// TwinCAT 3 PLC project ApplicationBase
// Title: ApplicationBase
// Company: Beckhoff Automation LLC
// Author: FS
// ProjectVersion: 2.3.0
// Description: All sample code provided by Beckhoff Automation LLC are for illustrative purposes only and are provided “as is” and without any warranties, express or implied. Actual implementations in applications will vary significantly. Beckhoff Automation LLC shall have no liability for, and does not waive any rights in relation to, any code samples that it provides or the use of such code samples for any purpose.
// ProgramVersion: 3.1.4026.27
// libraries:
//   Tc2_DataExchange, * (Beckhoff Automation GmbH)
//   Tc2_EtherCAT, * (Beckhoff Automation GmbH)
//   Tc2_IoFunctions, * (Beckhoff Automation GmbH)
//   Tc2_Math, * (Beckhoff Automation GmbH)
//   Tc2_MC2, * (Beckhoff Automation GmbH)
//   Tc2_MC2_Camming, * (Beckhoff Automation GmbH)
//   Tc2_MC2_Drive, * (Beckhoff Automation GmbH)
//   Tc2_NcKinematicTransformation, * (Beckhoff Automation GmbH)
//   Tc2_SerialCom, * (Beckhoff Automation GmbH)
//   Tc2_Standard, * (Beckhoff Automation GmbH)
//   Tc2_System, * (Beckhoff Automation GmbH)
//   Tc2_TcpIp, * (Beckhoff Automation GmbH)
//   Tc2_Utilities, * (Beckhoff Automation GmbH)
//   Tc3_DynamicMemory, * (Beckhoff Automation GmbH)
//   Tc3_EventLogger, * (Beckhoff Automation GmbH)
//   Tc3_JsonXml, * (Beckhoff Automation GmbH)
//   Tc3_MC2_AdvancedHoming, * (Beckhoff Automation GmbH)
//   Tc3_Mc3Ptp, * (Beckhoff Automation GmbH)
//   Tc3_Module, * (Beckhoff Automation GmbH)
//   Tc3_PackML_V3, * (Beckhoff Automation GmbH)
// project tree:
//   Components/ADS/ AdsReadWrite.TcPOU
//   Components/ADS/Interface/ I_AdsAccess.TcIO, I_AdsRW.TcIO
//   Components/Analog/ AnalogInput.TcPOU, AnalogInput_Generic.TcPOU, AnalogInput_Standard.TcPOU, AnalogOutput.TcPOU
//   Components/Analog/DUT/ ST_AnalogInputStatus_EL30xx.TcDUT, ST_AnalogInputStatus_Generic.TcDUT
//   Components/Analog/Interface/ I_AnalogChannel_Generic.TcIO, I_AnalogChannel_Standard.TcIO, I_AnalogInput.TcIO, I_AnalogOutput.TcIO
//   Components/CoE/ CoeDevice.TcPOU, NullCoeDevice.TcPOU
//   Components/CoE/DUT/ ST_TerminalProductInfo.TcDUT
//   Components/CoE/Interface/ I_CoeAccess.TcIO, I_CoeDevice.TcIO, I_CoeTransfer.TcIO, I_CoeTransferScheduler.TcIO
//   Components/Cylinder/ Cylinder.TcPOU, Cylinder_HMI.TcPOU, Cylinder_TcEvents.TcPOU
//   Components/Cylinder/DUT/ E_CylinderErrorId.TcDUT, E_CylinderState.TcDUT, ST_Cylinder_HMI.TcDUT
//   Components/Cylinder/Interface/ I_Cylinder.TcIO, I_CylinderCommand.TcIO, I_CylinderStatus.TcIO
//   Components/Digital/ DigitalInput_Combiner.TcPOU, DigitalInput_DebounceFallingEdge.TcPOU, DigitalInput_DebounceRisingEdge.TcPOU, DigitalInput_HMI.TcPOU, DigitalInput_NC.TcPOU, DigitalInput_NO.TcPOU, DigitalOutput.TcPOU, DigitalOutput_HMI.TcPOU
//   Components/Digital/DUT/ ST_DigitalInput_HMI.TcDUT, ST_DigitalOutput_HMI.TcDUT
//   Components/Digital/Interface/ I_DigitalInput.TcIO, I_DigitalOutput.TcIO
//   Components/Digital/Visitor/ ForceVisitor.TcPOU, ReleaseAllForceVisitor.TcPOU
//   Components/EtherCat/DUT/ E_EcErrorSource.TcDUT, EtherCatParameter.TcGVL, ST_EtherCatMasterInfo.TcDUT, ST_EtherCatSyncUnitTaskInfo.TcDUT
//   Components/EtherCat/ EtherCatIoDevice.TcPOU, EtherCatMaster.TcPOU, EtherCatMaster_TcEvents.TcPOU, SyncUnitTask.TcPOU
//   Components/EtherCat/Interface/ I_EcIoDevice.TcIO, I_EcSlaveRegistry.TcIO, I_EtherCatDiagnosticEventProvider.TcIO, I_EtherCatMasterDiagnostic.TcIO, I_IoDevice.TcIO, I_SyncUnitTask.TcIO
//   Components/Recipe/Interface/ I_RecipeManagment.TcIO
//   Components/Recipe/ RecipeManagment.TcPOU
//   Components/Safety/DUT/ E_SafetyConnection_State.TcDUT, E_SafetyEdm_State.TcDUT, E_SafetyEStop_State.TcDUT, E_SafetyGroup_Diag.TcDUT, E_SafetyGroup_State.TcDUT, E_SafetyMon_State.TcDUT, E_SafetyOrAnd_State.TcDUT, ST_SafetyAddressInfo.TcDUT, ST_SafetyDeviceInfo.TcDUT, ST_SafetyStateDiag.TcDUT
//   Components/Safety/Interface/ I_InSafetyGroup.TcIO, I_SafetyBase.TcIO, I_SafetyModule.TcIO, I_SafetyReset.TcIO, I_SafetySimulation.TcIO
//   Components/Safety/Reset Function/ SafetyResetPulse.TcPOU
//   Components/Safety/ SafetyAndOrFB.TcPOU, SafetyBase.TcPOU, SafetyConnectionFB_TcEvents.TcPOU, SafetyEdmFB_TcEvents.TcPOU, SafetyEstopFB_TcEvents.TcPOU, SafetyGroup_TcEvents.TcPOU, SafetyModule.TcPOU, SafetyMonFB_TcEvents.TcPOU
//   Components/Safety/Visitor/ SafetyOkVisitor.TcPOU, SetSafetySimulationVisitor.TcPOU
//   Components/Serial/Interface/ I_SerialByteConnection.TcIO, I_SerialLineControl.TcIO, I_SerialStringConnection.TcIO
//   Components/Serial/ SerialByteConnection.TcPOU, SerialLineControl_ADS.TcPOU, SerialLineControl_Terminal.TcPOU, SerialStringConnection.TcPOU
//   Components/Tcp Ip/DUT/ ST_TcpIpPayload.TcDUT
//   Components/Tcp Ip/Interface/ I_TcpIpConnection.TcIO, I_TcpIpSubscription.TcIO
//   Components/Tcp Ip/ TcpIpCommandResultFilter.TcPOU, TcpIpConnection.TcPOU, TcpIpConnectionParameter.TcGVL
//   Component/ Component.TcPOU, CyclicComponent.TcPOU
//   Component/Interface/ I_Component.TcIO, I_ComponentVisitor.TcIO
//   / ApplicationBaseParameter.TcGVL, ApplicationBaseMotionParameter.TcGVL
//   Events/Interface/ I_EventArguments.TcIO, I_EventClass.TcIO, I_EventClassTcEvents.TcIO, I_EventReaction.TcIO, I_EventReactionTcEvents.TcIO
//   Events/ TcEventClass.TcPOU
//   HMI/ Button.TcPOU, HmiFunction.TcPOU
//   HMI/DUT/ ST_HmiFunction.TcDUT
//   HMI/Interface/ I_Button.TcIO, I_HmiFunction.TcIO, I_Permissive.TcIO, I_StringCollection.TcIO
//   Kinematic Group/Interface/ I_KinematicGroup.TcIO
//   Kinematic Group/ KinematicGroup.TcPOU, KinematicGroup_TcEvents.TcPOU
//   Modes/Interface/ I_Mode.TcIO
//   Modes/ ModeControl.TcPOU, PackMLModeControl.TcPOU
//   Module PackML/ PackMLModule.TcPOU
//   Module/Interface/ I_Module.TcIO, I_ModuleVisitor.TcIO
//   Module/ Module.TcPOU
//   Motion/ AxisPTP_HMI.TcPOU, Axis_TcEvents.TcPOU
//   Motion/DUT/ E_AxisJogMode.TcDUT, ST_AxisPTP_HMI.TcDUT, ST_NcAxisStatus.TcDUT
//   Motion/Interface/ I_AxisDynamics.TcIO, I_AxisEnable.TcIO, I_AxisHome.TcIO, I_AxisJog.TcIO, I_AxisMoveAbsolute.TcIO, I_AxisMoveModulo.TcIO, I_AxisMoveRelative.TcIO, I_AxisMoveVelocity.TcIO, I_AxisStatus.TcIO, I_Axis.TcIO, I_AxisGear.TcIO, I_AxisSettings.TcIO, I_Axis_PTP.TcIO, I_MotionTaskCollection.TcIO
//   Motion/MC2/DUT/ ST_Mc2MotionDefaults.TcDUT
//   Motion/MC2/Interface/ I_Mc2Axis.TcIO, I_Mc2AxisGear.TcIO, I_Mc2Axis_PTP.TcIO, I_Mc2Settings.TcIO, I_Mc2SlaveAxis.TcIO
//   Motion/MC2/ Mc2Axis.TcPOU, Mc2AxisPTP.TcPOU, Mc2AxisParameterLoader.TcPOU, Mc2SlaveAxisPTP.TcPOU
//   Motion/MC3/DUT/ ST_Mc3MotionDefaults.TcDUT, ST_Mc3ParameterBinding.TcDUT
//   Motion/MC3/Interface/ I_Mc3SlaveAxis.TcIO, I_Mc3AxisGear.TcIO, I_Mc3Axis_PTP.TcIO, I_Mc3Settings.TcIO, I_Mc3Axis.TcIO
//   Motion/MC3/ Mc3SlaveAxisPTP.TcPOU, Mc3AxisPTP.TcPOU, Mc3AxisParameterLoader.TcPOU, Mc3Axis.TcPOU
//   Permissive Interlock/ PermissiveInterlock.TcPOU
//   Project Information/ F_GetCompany.TcPOU, F_GetTitle.TcPOU, F_GetVersion.TcPOU
//   Statemachine/DUT/ ST_PackMLStatemachine_HMI.TcDUT, ST_Statemachine_HMI.TcDUT
//   Statemachine/Generic/ NextMinorStep.TcPOU (not stored), NextStep.TcPOU (not stored), SetStep.TcPOU (not stored), State.TcPOU, Statemachine.TcPOU, Statemachine_HMI.TcPOU
//   Statemachine/Interface/ I_ContainStatemachine.TcIO, I_State.TcIO, I_Statemachine.TcIO
//   Statemachine/PackML/ NextAvailablePackMLCommands.TcPOU (not stored), PackMLStatemachine.TcPOU, PackMLStatemachine_HMI.TcPOU, PackMLStatemachine_ModuleIntegrated.TcPOU
//   Tracing/ CoreTrace.TcGVL, Trace.TcPOU
//   Tracing/DUT/ TcEventSeverityExt.TcDUT (not stored)
//   Tracing/Interface/ I_Trace.TcIO (not stored)
//   Utilities/AnyBuffer/ AnyBuffer.TcPOU
//   Utilities/AnyBuffer/DUT/ ST_BufferConfiguration.TcDUT, ST_BufferMetadata.TcDUT
//   Utilities/AnyBuffer/Interface/ I_AnyBuffer.TcIO, I_AnyBufferStrategy.TcIO
//   Utilities/AnyBuffer/TypedBuffers/ FifoBuffer.TcPOU, LifoBuffer.TcPOU, ListBuffer.TcPOU, RingBuffer.TcPOU
//   Utilities/File/DUT/ ST_File_HMI.TcDUT
//   Utilities/File/ File_HMI.TcPOU, JsonFile.TcPOU, StringHelper.TcPOU
//   Utilities/File/Interface/ I_FileHandler.TcIO
//   Utilities/Flash/ SyncedSquareWaves.TcPOU
//   Utilities/Force/DUT/ E_ForceState.TcDUT
//   Utilities/Force/ ForcibleBool.TcPOU, ForcibleInt.TcPOU
//   Utilities/Force/Interface/ I_ForcibleBool.TcIO, I_ForcibleInt.TcIO
//   Utilities/Functions/ CompareLREAL.TcPOU, CompareModulo.TcPOU, PercentToAnalog.TcPOU
//   Utilities/Motion/ ATAN2.TcPOU, CalculateHypotenuseAngle.TcPOU, CalculateMotionDynamics.TcPOU, CamSmoothError.TcDUT, CamSplineBoundary.TcDUT, CamSmoothDerivatives.TcPOU, MotionDynamicsError.TcDUT, XPlanar6DMoverToWorldTransform.TcPOU
//   Utilities/Scaling/ AnalogScale.TcPOU, Calibrate.TcPOU
//   Utilities/Scaling/Interface/ I_AnalogScalable.TcIO, I_AnalogScale.TcIO, I_CalibratableLinear.TcIO, I_CalibrateLinear.TcIO, I_TransformLRealValue.TcIO
//   Utilities/Timing/ Stopwatch.TcPOU
//   Version/ Global_Version.TcGVL
//   Visitors/Enable/ CheckComponentsEnabledVisitor.TcPOU, DisableAllComponentsVisitor.TcPOU, EnableAllComponentsVisitor.TcPOU
//   Visitors/Events/ GetActiveEventSeverityVisitor.TcPOU
//   Visitors/HMI/ GetSystemTreeJsonHmiVisitor.TcPOU, HmiEnableDisableAllVisitor.TcPOU
//   Visitors/Override/ SetAllOverrideVisitor.TcPOU
//   Visitors/PackML Statemachine/ ChangePackMLStateOnAllSubModulesVisitor.TcPOU, EventReactorPackMLVisitor.TcPOU
//   Visitors/Reset/ GetComponentsTaskResultVisitor.TcPOU, ResetAllVisitor.TcPOU, ResetComponentsVisitor.TcPOU, ResetModulesVisitor.TcPOU
//   Visitors/Statemachine/ ChangeModeOnAllSubModulesVisitor.TcPOU, ChangeStateOnAllSubModulesVisitor.TcPOU, EventReactorVisitor.TcPOU
//   Visitors/Stop/ StopAllComponentsVisitor.TcPOU
//   _Interface/ I_Base.TcIO (not stored), I_Command.TcIO, I_Disposable.TcIO, I_Enablable.TcIO, I_Initializable.TcIO, I_Override.TcIO, I_Resettable.TcIO, I_Simulatable.TcIO, I_Stoppable.TcIO, I_TaskResult.TcIO, I_ToString.TcIO (not stored)
//   _Internal/CollectionPeeker/ CollectionPeeker.TcPOU
//   _Internal/CollectionPeeker/Interface/ I_CollectionPeeker.TcIO, I_Peekable.TcIO, I_Peeker.TcIO
//   _Internal/Collection/ Collection.TcPOU
//   _Internal/Collection/Interface/ I_Collection.TcIO, I_Enumerator.TcIO
//   _Internal/Component/ ComponentCollection.TcPOU
//   _Internal/Component/Interface/ I_ComponentCollection.TcIO, I_ContainComponents.TcIO
//   _Internal/Cyclic/ CyclicRunner.TcPOU
//   _Internal/Cyclic/Interface/ I_Cyclic.TcIO
//   _Internal/Events/ TcEventClassArguments.TcPOU
//   _Internal/Initialize/ Initializer.TcPOU
//   _Internal/List/Interface/ I_List.TcIO
//   _Internal/List/ List.TcPOU
//   _Internal/Module/Interface/ I_ContainModules.TcIO, I_ModuleCollection.TcIO
//   _Internal/Module/ ModuleCollection.TcPOU
//   _Internal/MotionTasks/DUT/ ST_TaskState.TcDUT
//   _Internal/MotionTasks/MC2/AX5000/DUT/P_0_0074/ ST_IDN_P_0_0074.TcDUT (not stored), ST_IDN_P_0_0074_UDINT.TcDUT
//   _Internal/MotionTasks/MC2/AX5000/DUT/P_0_0074_LREAL/ ST_IDN_P_0_0074_LREAL.TcDUT
//   _Internal/MotionTasks/MC2/AX5000/DUT/ ST_AX5000AmpToNm.TcDUT
//   _Internal/MotionTasks/MC2/AX5000/ Mc2MotionTask_AX5000AmpToNm.TcPOU
//   _Internal/MotionTasks/MC2/Base/ Mc2MotionTask.TcPOU, Mc2MotionTaskCollection.TcPOU
//   _Internal/MotionTasks/MC2/Coupling/ Mc2MotionCoupleTask_Gearing.TcPOU
//   _Internal/MotionTasks/MC2/Home/ Mc2MotionHomeTask_CoESetEncoderOffset.TcPOU, Mc2MotionHomeTask_SetPosition.TcPOU, Mc2MotionHomeTask_SetPositionOffset.TcPOU, Mc2MotionHomeTask_SetZeroHere.TcPOU, Mc2MotionHomeTask_TouchProbe.TcPOU
//   _Internal/MotionTasks/MC2/Interface/ I_Mc2AxisRef.TcIO, I_Mc2MotionJogTask.TcIO, I_Mc2MotionPowerTask.TcIO, I_Mc2MotionTask.TcIO, I_Mc2MotionTaskCollection.TcIO
//   _Internal/MotionTasks/MC2/Move/ Mc2MoveAbsoluteTask.TcPOU, Mc2MoveJogTask.TcPOU, Mc2MoveModuloTask.TcPOU, Mc2MoveRelativeTask.TcPOU, Mc2MoveVelocityTask.TcPOU
//   _Internal/MotionTasks/MC2/Power/ Mc2PowerTask.TcPOU, Mc2StopTask.TcPOU
//   _Internal/MotionTasks/MC2/Reset/ Mc2CoEExtendedResetTask.TcPOU, Mc2CoEResetTask.TcPOU, Mc2SoEResetTask.TcPOU
//   _Internal/MotionTasks/MC3/Base/ Mc3MotionTaskCollection.TcPOU, Mc3MotionTask.TcPOU
//   _Internal/MotionTasks/MC3/Gearing/ Mc3MotionCoupleTask_Gearing.TcPOU
//   _Internal/MotionTasks/MC3/Home/ Mc3MotionHomeTask_SetPosition.TcPOU, Mc3MotionHomeTask_SetZeroHere.TcPOU
//   _Internal/MotionTasks/MC3/Interface/ I_Mc3AxisRef.TcIO, I_Mc3MotionJogTask.TcIO, I_Mc3MotionPowerTask.TcIO, I_Mc3MotionTaskCollection.TcIO, I_Mc3MotionTask.TcIO
//   _Internal/MotionTasks/MC3/Move/ Mc3MoveAbsoluteTask.TcPOU, Mc3MoveModuloTask.TcPOU, Mc3MoveRelativeTask.TcPOU, Mc3MoveVelocityTask.TcPOU, Mc3MoveJogTask.TcPOU
//   _Internal/MotionTasks/MC3/Power/ Mc3PowerTask.TcPOU, Mc3StopTask.TcPOU
//   _Internal/MotionTasks/MC3/Reset/ Mc3CoEResetTask.TcPOU
//   _Internal/Null/ NullComponent.TcPOU, NullItem.TcPOU, NullModule.TcPOU
//   _Internal/Statemachine/Interface/ I_StateList.TcIO
//   _Internal/Statemachine/ StateList.TcPOU
//   _Internal/Tracing/ AdsLogger.TcPOU, LocalLogger.TcPOU, TcEventLogger.TcPOU, TraceMessageInfo.TcPOU, TraceSourceInfo.TcPOU, USINT_To_TcEventSeverity.TcPOU (not stored)
//   _Internal/Tracing/Interface/ I_ContainTraceArgument.TcIO (not stored), I_ContainTracePublisher.TcIO (not stored), I_TraceArgument.TcIO, I_TraceInstanceLogger.TcIO (not stored), I_TraceLogger.TcIO (not stored), I_TraceMessageInfo.TcIO (not stored), I_TracePublisher.TcIO (not stored), I_TraceSourceInfo.TcIO (not stored)
//   _Internal/Types/ RegistrationResult.TcDUT

// ---- Components/Analog/DUT/ST_AnalogInputStatus_EL30xx.TcDUT
{attribute 'pack_mode' := '1'}
TYPE ST_AnalogInputStatus_EL30xx :
	STRUCT
		Underrrange : BIT;
		Overrange	: BIT;
		Limit1L		: BIT;
		Limit1H		: BIT;
		Limit2L		: BIT;
		Limit2H		: BIT;
		Error		: BIT;
		TxPDOState	: BIT;
		TxPDOToggle : BIT;
	END_STRUCT
END_TYPE

// ---- Components/Analog/DUT/ST_AnalogInputStatus_Generic.TcDUT
{attribute 'pack_mode' := '1'}
TYPE ST_AnalogInputStatus_Generic :
	STRUCT
		Underrrange : BIT;
		Overrange	: BIT;
		Error		: BIT;
		WcState		: BIT;
	END_STRUCT
END_TYPE

// ---- Components/CoE/DUT/ST_TerminalProductInfo.TcDUT
{attribute 'pack_mode' := '2'}
TYPE ST_TerminalProductInfo : // Parameter 16#1018:0
	STRUCT
		Identity	 : WORD;
		VendorId	 : DINT;
		ProductCode	 : DINT;
		Revision	 : DINT;
		SerialNumber : DINT;
	END_STRUCT
END_TYPE

// ---- Components/Cylinder/DUT/E_CylinderErrorId.TcDUT
{attribute 'qualified_only'}
TYPE E_CylinderErrorId : (
		NoError				  := 0,
		ExtendTimeout		  := 1,
		RetractTimeout		  := 2,
		ExtendedPlausibility  := 3,
		RetractedPlausibility := 4,
		BothSensorsActive	  := 5
	) UDINT;
END_TYPE

// ---- Components/Cylinder/DUT/E_CylinderState.TcDUT
{attribute 'qualified_only'}
TYPE E_CylinderState : (
		Undefined  := 0,
		Extending  := 1,
		Extended   := 2,
		Retracting := 3,
		Retracted  := 4
	);
END_TYPE

// ---- Components/Cylinder/DUT/ST_Cylinder_HMI.TcDUT
TYPE ST_Cylinder_HMI EXTENDS ST_HmiFunction :
	STRUCT
		Busy		  : BOOL;
		Error		  : BOOL;
		ErrorId		  : UDINT;
		Extended	  : BOOL;
		ExtendedName  : STRING := 'Extended';
		Retracted	  : BOOL;
		RetractedName : STRING := 'Retracted';
		Extend		  : Button;
		Retract		  : Button;
	END_STRUCT
END_TYPE

// ---- Components/Digital/DUT/ST_DigitalInput_HMI.TcDUT
TYPE ST_DigitalInput_HMI EXTENDS ST_HmiFunction :
	STRUCT
		Active : BOOL;
		Force  : E_ForceState;
	END_STRUCT
END_TYPE

// ---- Components/Digital/DUT/ST_DigitalOutput_HMI.TcDUT
TYPE ST_DigitalOutput_HMI EXTENDS ST_HmiFunction :
	STRUCT
		On	  : BOOL;
		Force : E_ForceState;
	END_STRUCT
END_TYPE

// ---- Components/EtherCat/DUT/E_EcErrorSource.TcDUT
{attribute 'qualified_only'}
{attribute 'strict'}
// Origin of EtherCatMaster.ErrorId. ErrorId keeps the raw code of that source:
//   Master   - EcMaster.DevState word
//   Slave    - configured slave index (0-based, configuration order)
//   Ads      - error id of the Tc2_EtherCAT / ADS function block (16#745 = watchdog timeout)
//   Sequence - step number or count that violated a precondition
TYPE E_EcErrorSource :
(
	None	 := 0,
	Master	 := 1,
	Slave	 := 2,
	Ads		 := 3,
	Sequence := 4
) UINT;
END_TYPE

// ---- Components/EtherCat/DUT/ST_EtherCatMasterInfo.TcDUT
TYPE ST_EtherCatMasterInfo :
	STRUCT
		AmsNetID	  : AMSNETID;
		DevID		  : UINT;
		DevState	  : UINT;
		ChangeCount	  : UINT;
		SlaveCount	  : UINT;
		CfgSlaveCount : UINT;
	END_STRUCT
END_TYPE

// ---- Components/EtherCat/DUT/ST_EtherCatSyncUnitTaskInfo.TcDUT
TYPE ST_EtherCatSyncUnitTaskInfo :
	STRUCT
		WcState	   : BIT;
		ObjectId   : OTCID;
		State	   : UINT;
		SlaveCount : UINT;
	END_STRUCT
END_TYPE

// ---- Components/Safety/DUT/E_SafetyConnection_State.TcDUT
{attribute 'qualified_only'}
{attribute 'strict'}
TYPE E_SafetyConnection_State : (
		Reset	   := 100,
		Session	   := 101,
		Connection := 102,
		Parameter  := 103,
		Data	   := 104,
		Shutdown   := 105,
		Deactive   := 106
	) USINT;
END_TYPE

// ---- Components/Safety/DUT/E_SafetyEdm_State.TcDUT
{attribute 'qualified_only'}
TYPE E_SafetyEdm_State : (
		Invalid := 0,
		Stop	:= 2,
		Error	:= 4,
		Reset	:= 5,
		MonOff	:= 14,
		MonOn	:= 15
	) USINT;
END_TYPE

// ---- Components/Safety/DUT/E_SafetyEStop_State.TcDUT
{attribute 'qualified_only'}
TYPE E_SafetyEStop_State : (
		Invalid	 := 0,
		Run		 := 1,
		Stop	 := 2,
		Safe	 := 3,
		Error	 := 4,
		Reset	 := 5,
		Start	 := 6,
		DelayOut := 7
	) USINT;
END_TYPE

// ---- Components/Safety/DUT/E_SafetyGroup_Diag.TcDUT
{attribute 'qualified_only'}
TYPE E_SafetyGroup_Diag : (
		NoError		  := 0,
		FbError		  := 1,
		ComError	  := 2,
		ModuleError	  := 3,
		CmpError	  := 4,
		DeactiveError := 5,
		RestartError  := 6
	) UINT;
END_TYPE

// ---- Components/Safety/DUT/E_SafetyGroup_State.TcDUT
{attribute 'qualified_only'}
TYPE E_SafetyGroup_State : (
		Invalid		 := 0,
		Run			 := 1,
		Stop		 := 2,
		Error		 := 4,
		Reset		 := 5,
		Start		 := 6,
		StopError	 := 7,
		Deactive	 := 16,
		WaitComError := 17
	) USINT;
END_TYPE

// ---- Components/Safety/DUT/E_SafetyMon_State.TcDUT
{attribute 'qualified_only'}
TYPE E_SafetyMon_State : (
		Invalid	   := 0,
		Run		   := 1,
		Stop	   := 2,
		Safe	   := 3,
		Error	   := 4,
		Reset	   := 5,
		Start	   := 6,
		ErrorDelay := 7,
		DelayOut   := 8,
		FuncTest   := 9
	) USINT;
END_TYPE

// ---- Components/Safety/DUT/E_SafetyOrAnd_State.TcDUT
{attribute 'qualified_only'}
TYPE E_SafetyOrAnd_State : (
		Invalid := 0,
		Run		:= 1,
		Stop	:= 2,
		Safe	:= 3
	) USINT;
END_TYPE

// ---- Components/Safety/DUT/ST_SafetyAddressInfo.TcDUT
{attribute 'pack_mode' := '2'}
TYPE ST_SafetyAddressInfo : // Parameter 16#F980:0
	STRUCT
		FSoEAddress		  : WORD;
		SerialNumber	  : DINT;
		ProjectCRC		  : WORD;
		DefaultProjectCRC : WORD;
	END_STRUCT
END_TYPE

// ---- Components/Safety/DUT/ST_SafetyDeviceInfo.TcDUT
{attribute 'pack_mode' := '2'}
TYPE ST_SafetyDeviceInfo : // Parameter 16#F9C0:0
	STRUCT
		DeviceName			 : STRING;
		SoftwareVersion		 : STRING;
		BootloaderVersion	 : STRING;
		SoftwareChecksum	 : DINT;
		BootmanagerChecksum	 : DINT;
		BootloaderChecksum	 : DINT;
		TwinSAFELogicVersion : DINT;
	END_STRUCT
END_TYPE

// ---- Components/Safety/DUT/ST_SafetyStateDiag.TcDUT
{attribute 'pack_mode' := '1'}
TYPE ST_SafetyStateDiag :
	STRUCT
		State : USINT;
		Diag  : UINT; // **NOT PRESENT ON AND/OR FBs ** For components with USINT as Diag connection, connect first 8 Bit of UINT Diag. Inherited FB is evaluating correct length.
	END_STRUCT
END_TYPE

// ---- Components/Tcp Ip/DUT/ST_TcpIpPayload.TcDUT
TYPE ST_TcpIpPayload :
	STRUCT
		Size : UDINT;
		Data : ARRAY[0..(TcpIpConnectionParameter.PayloadSize - 1)] OF BYTE;
	END_STRUCT
END_TYPE

// ---- HMI/DUT/ST_HmiFunction.TcDUT
TYPE ST_HmiFunction :
	STRUCT
		Name	   : STRING;
		HmiEnabled : BOOL := TRUE;
	END_STRUCT
END_TYPE

// ---- Motion/DUT/E_AxisJogMode.TcDUT
{attribute 'qualified_only'}
{attribute 'strict'}
(* Motion-generation independent jog mode.
   Mapped onto Tc2_MC2.E_JogMode / Tc3_Mc3Ptp.EJogMode by the concrete axis. *)
TYPE E_AxisJogMode : (
		Slow := 0,
		Fast := 1
	) DINT;
END_TYPE

// ---- Motion/DUT/ST_AxisPTP_HMI.TcDUT
TYPE ST_AxisPTP_HMI EXTENDS ST_HmiFunction :
	STRUCT
		Unit				 : STRING;
		Busy				 : BOOL;
		Error				 : BOOL;
		ErrorId				 : UDINT;
		ActualAcceleration	 : LREAL;
		ActualPosition		 : LREAL;
		ActualPositionModulo : LREAL;
		ActualTorque		 : LREAL;
		ActualVelocity		 : LREAL;
		Status				 : ST_NcAxisStatus;
		Enable				 : Button;
		Disable				 : Button;
		Stop				 : Button;
		JogForwardSlow		 : Button;
		JogBackwardSlow		 : Button;
		JogForwardFast		 : Button;
		JogBackwardFast		 : Button;
		Home				 : Button;
		Reset				 : Button;
		MoveAbsolute		 : Button;
		TargetPosition		 : LREAL;
		MoveVelocity		 : Button;
		TargetVelocity		 : LREAL;
		MoveRelative		 : Button;
		TargetDistance		 : LREAL;
		MoveModulo			 : Button;
	END_STRUCT
END_TYPE

// ---- Motion/DUT/ST_NcAxisStatus.TcDUT
TYPE ST_NcAxisStatus :
	STRUCT
		Disabled		   : BOOL;
		SynchronizedMotion : BOOL;
		Coupled			   : BOOL;
	END_STRUCT
END_TYPE

// ---- Motion/MC2/DUT/ST_Mc2MotionDefaults.TcDUT
TYPE ST_Mc2MotionDefaults :
	STRUCT
		DefaultResetTask : Mc2CoEResetTask				 := (Name := 'MC Reset (CoE)');
		DefaultHomeTask	 : Mc2MotionHomeTask_SetZeroHere := (Name := 'MC Home');
		DefaultStopTask	 : Mc2StopTask					 := (Name := 'MC Stop');
	END_STRUCT
END_TYPE

// ---- Motion/MC3/DUT/ST_Mc3MotionDefaults.TcDUT
TYPE ST_Mc3MotionDefaults :
	STRUCT
		DefaultResetTask : Mc3CoEResetTask				 := (Name := 'MC Reset (CoE)');
		DefaultHomeTask	 : Mc3MotionHomeTask_SetZeroHere := (Name := 'MC Home');
		DefaultStopTask	 : Mc3StopTask					 := (Name := 'MC Stop');
	END_STRUCT
END_TYPE

// ---- Motion/MC3/DUT/ST_Mc3ParameterBinding.TcDUT
(* One entry in an Mc3AxisParameterLoader table: which NC axis parameter to
   read, and where in the owning axis to store it. *)
TYPE ST_Mc3ParameterBinding :
STRUCT
	ParameterId : Tc3_Mc3Ptp.EAxisParameterId;
	Target		: POINTER TO LREAL;
END_STRUCT
END_TYPE

// ---- Statemachine/DUT/ST_PackMLStatemachine_HMI.TcDUT
TYPE ST_PackMLStatemachine_HMI EXTENDS ST_HmiFunction :
	STRUCT
		// Simplified Control
		ResetPermissive : BOOL;
		ResetPressed	: BOOL;
		Resetted		: BOOL;
		StartPermissive : BOOL;
		StartPressed	: BOOL;
		Started			: BOOL;
		StopPermissive	: BOOL;
		StopPressed		: BOOL;
		Stopped			: BOOL;
		// Standard Control
		CurrentMode	 : DINT;
		ModeCommand	 : DINT;
		CurrentState : E_PMLState;
		StateCommand : E_PMLCommand;
		// Next Available Commands
		NextAvailableCommands : ARRAY[0..9] OF E_PMLCommand;
	END_STRUCT
END_TYPE

// ---- Statemachine/DUT/ST_Statemachine_HMI.TcDUT
TYPE ST_Statemachine_HMI EXTENDS ST_HmiFunction :
	STRUCT
		CurrentState	   : DINT;
		CurrentMode		   : DINT;
		StateChangeCommand : DINT;
		ModeChangeCommand  : DINT;
	END_STRUCT
END_TYPE

// ---- Utilities/AnyBuffer/DUT/ST_BufferConfiguration.TcDUT
TYPE ST_BufferConfiguration :
	STRUCT
		isPersistent	 : BOOL; // is the buffer persistent?
		capacity		 : DINT; // No of elements in buffer
		elementSize		 : DINT; // Buffer element size in bytes
		bufferSize		 : DINT; // Complete buffer size in bytes	
		bufferBoundLower : DINT; // Lower boundary of the buffer
		bufferBoundUpper : DINT; // Upper boundary of the buffer	
	END_STRUCT
END_TYPE

// ---- Utilities/AnyBuffer/DUT/ST_BufferMetadata.TcDUT
TYPE ST_BufferMetadata :
	STRUCT
		headIndex	 : DINT;
		tailIndex	 : DINT;
		capacity	 : DINT;
		elementCount : DINT;
	END_STRUCT
END_TYPE

// ---- Utilities/File/DUT/ST_File_HMI.TcDUT
TYPE ST_File_HMI EXTENDS ST_HmiFunction :
	STRUCT
		Path	: STRING;
		Load	: Button;
		Save	: Button;
		NewPath : BOOL;
	END_STRUCT
END_TYPE

// ---- Utilities/Force/DUT/E_ForceState.TcDUT
{attribute 'qualified_only'}
{attribute 'strict'}
{attribute 'to_string'}
TYPE E_ForceState : (
		Unforced := 0,
		ForceOn	 := 1,
		ForceOff := 2
	) DINT;
END_TYPE

// ---- Utilities/Motion/CamSmoothError.TcDUT
TYPE CamSmoothError :
(
    NoError            := 0,
    RangeOutsideArray  := 1,    // nFirst / nLast not inside aPoints
    TooFewPoints       := 2,    // fewer than 4 points in the range
    TooManyPoints      := 3,    // range exceeds GVL_Cam.CAM_MAX_POINTS
    BadDecimals        := 4,    // nDecimals outside 0..9
    MasterNotAscending := 5,    // MasterPos must strictly increase
    SolverSingular     := 6     // zero pivot in the tridiagonal solve
)
INT;
END_TYPE

// ---- Utilities/Motion/CamSplineBoundary.TcDUT
TYPE CamSplineBoundary :
(
    // 3rd derivative continuous across the 2nd and 2nd-last knot, so the
    // spline follows the profile's own curvature at the ends.
    // General-purpose default.
    NotAKnot := 0,

    // SlaveAcc forced to 0.0 at the first and last profile point.
    // Use when the axis enters and leaves the profile with no acceleration,
    // e.g. when a POLYNOM1 ramp sits on either side of the profile.
    Natural  := 1
)
INT;
END_TYPE

// ---- Utilities/Motion/MotionDynamicsError.TcDUT
{attribute 'qualified_only'}
{attribute 'strict'}
TYPE MotionDynamicsError :
(
    /// No error, the calculated dynamics are valid
    NoError := 0,
    /// ABS(Distance) is zero (or not a usable number) - nothing to move
    InvalidDistance := 1,
    /// MoveTime is zero or negative
    InvalidMoveTime := 2,
    /// VelocityMax is zero or negative
    InvalidVelocityMax := 3,
    /// AccelerationMax is zero or negative
    InvalidAccelerationMax := 4,
    /// DecelerationMax is zero or negative
    InvalidDecelerationMax := 5,
    /// JerkMax is negative (0 is allowed and means "no jerk limitation")
    InvalidJerkMax := 6,
    /// MoveTime is shorter than the fastest possible move (TimeMin).
    /// The outputs still contain the fastest feasible profile (= the maximum dynamics).
    TimeTooShort := 7,
    /// Internal solver did not return a usable peak velocity
    CalculationFailed := 8
) DINT;
END_TYPE

// ---- _Internal/MotionTasks/DUT/ST_TaskState.TcDUT
TYPE ST_TaskState :
	STRUCT
		Name	: T_MaxString;
		Busy	: BOOL;
		Error	: BOOL;
		ErrorId : UDINT;
	END_STRUCT
END_TYPE

// ---- _Internal/MotionTasks/MC2/AX5000/DUT/P_0_0074/ST_IDN_P_0_0074_UDINT.TcDUT
TYPE ST_IDN_P_0_0074_UDINT :
	STRUCT
		Actual	 : UINT;
		_Max	 : UINT;
		Elements : ST_IDN_P_0_0074;
	END_STRUCT
END_TYPE

// ---- _Internal/MotionTasks/MC2/AX5000/DUT/P_0_0074_LREAL/ST_IDN_P_0_0074_LREAL.TcDUT
TYPE ST_IDN_P_0_0074_LREAL :
	STRUCT
		Iq : ARRAY[0..9] OF LREAL;
		M  : ARRAY[0..9] OF LREAL;
	END_STRUCT
END_TYPE

// ---- _Internal/MotionTasks/MC2/AX5000/DUT/ST_AX5000AmpToNm.TcDUT
TYPE ST_AX5000AmpToNm :
	STRUCT
		Curve	   : ST_IDN_P_0_0074_LREAL; // Contents read in from P-0-0074   ( scaled )
		ActCurrent : LREAL;					// Actual current in Amps           ( units := A )
		ActTorque  : LREAL;					// Actual torque in Newton Meters   ( units := Nm )
	END_STRUCT
END_TYPE

// ---- _Internal/Types/RegistrationResult.TcDUT
{attribute 'qualified_only'}
{attribute 'strict'}
{attribute 'to_string'}
TYPE RegistrationResult :
(
	Succeeded := 0,
	NullReference := -1,
	TooManyComponents := -2,
	AlreadyAdded := -3,
	CollectionEmpty := -4,
	NotFoundInCollection := -5
);
END_TYPE

// ---- Components/EtherCat/DUT/EtherCatParameter.TcGVL
VAR_GLOBAL CONSTANT
	// Upper index of every per-slave array in EtherCatMaster and SyncUnitTask; holds MAX_EC_SLAVES + 1 slaves.
	MAX_EC_SLAVES	 : UINT	 := 49;

	// Slaves handled per PLC cycle by the multi-cycle diagnostic passes (state classification, fault
	// evaluation, sync unit resolution). A pass over n slaves finishes within n / SLAVES_PER_CYCLE cycles.
	SLAVES_PER_CYCLE : UINT	 := 64;

	// Cycles a diagnostic ADS read may stay busy before the sequence aborts with E_EcErrorSource.Ads,
	// ErrorId 16#745 (1000 cycles = 10 s on a 10 ms task).
	ADS_WAIT_CYCLES	 : UDINT := 1000;

	// Cycles the one-off configuration and topology reads in Initialize may stay busy. Generous on purpose:
	// TwinCAT serves ADS reads above 128 KiB from a task that owns no process data on the master very slowly
	// (about 3 min for 2500 slaves).
	INIT_WAIT_CYCLES : UDINT := 60000;
END_VAR

// ---- Components/Tcp Ip/TcpIpConnectionParameter.TcGVL
{attribute 'qualified_only'}
VAR_GLOBAL CONSTANT
	PayloadSize : UDINT := 1460; // Payload in Bytes
END_VAR

// ---- ApplicationBaseParameter.TcGVL
{attribute 'qualified_only'}
VAR_GLOBAL CONSTANT
	MaxCountInCollections : UDINT			   := 50;
	EnableTcEventLogging  : BOOL			   := FALSE;
	EnableAdsLogger		  : BOOL			   := TRUE;
	ClearingTimeout		  : TIME			   := T#2S;
	TraceLevel			  : TcEventSeverityExt := TcEventSeverityExt.Verbose;
END_VAR

// ---- ApplicationBaseMotionParameter.TcGVL
{attribute 'qualified_only'}
VAR_GLOBAL CONSTANT
	MaxMotionTasks : UDINT := 10;
	// Upper bound for the NC parameter table each Mc3Axis pre-loads
	MaxAxisParameters : UDINT := 10;
END_VAR

// ---- Tracing/CoreTrace.TcGVL
VAR_GLOBAL
	Trace : Trace<ApplicationBaseParameter.MaxCountInCollections> := (TraceLevel := ApplicationBaseParameter.TraceLevel);
	{attribute 'hide'}
	TcEventLogger : TcEventLogger(Trace);
	{attribute 'hide'}
	AdsLogger : AdsLogger(Trace);
END_VAR

// ---- Version/Global_Version.TcGVL
{attribute 'TcGenerated'}
{attribute 'no-analysis'}
{attribute 'linkalways'}
// This function has been automatically generated from the project information.
VAR_GLOBAL CONSTANT
	{attribute 'const_non_replaced'}
	stLibVersion_ApplicationBase : ST_LibVersion := (iMajor := 2, iMinor := 3, iBuild := 0, iRevision := 0, nFlags := 0, sVersion := '2.3.0');
END_VAR

// ---- Components/ADS/Interface/I_AdsAccess.TcIO
INTERFACE I_AdsAccess EXTENDS I_Base

PROPERTY AdsRW : I_AdsRW
GET
END_GET
SET
END_SET
END_PROPERTY

END_INTERFACE

// ---- Components/ADS/Interface/I_AdsRW.TcIO
INTERFACE I_AdsRW EXTENDS I_Component, I_TaskResult

{attribute 'monitoring' := 'call'}
PROPERTY AmsNetId : T_AmsNetId
GET
END_GET
SET
END_SET
END_PROPERTY

{attribute 'monitoring' := 'call'}
PROPERTY AmsPort : T_AmsPort
GET
END_GET
SET
END_SET
END_PROPERTY

METHOD Read
VAR_INPUT
	IdxGrp	  : UDINT;
	IdxOffset : UDINT;
	pDestAddr : PVOID;
	Length	  : UDINT;
END_VAR
END_METHOD

METHOD ReadBySymbol
VAR_INPUT
	SymbolName : STRING(255);
	pDestAddr  : PVOID;
	Length	   : UDINT;
END_VAR
END_METHOD

METHOD Write
VAR_INPUT
	IdxGrp		: UDINT;
	IdxOffset	: UDINT;
	pSourceAddr : PVOID;
	Length		: UDINT;
END_VAR
END_METHOD

METHOD WriteBySymbol
VAR_INPUT
	SymbolName	: STRING(255);
	pSourceAddr : PVOID;
	Length		: UDINT;
END_VAR
END_METHOD

END_INTERFACE

// ---- Components/Analog/Interface/I_AnalogChannel_Generic.TcIO
INTERFACE I_AnalogChannel_Generic EXTENDS I_AnalogInput

PROPERTY DataValid : BOOL
GET
END_GET
END_PROPERTY

PROPERTY Error : BOOL
GET
END_GET
END_PROPERTY

PROPERTY Overrange : BOOL
GET
END_GET
END_PROPERTY

PROPERTY Underrange : BOOL
GET
END_GET
END_PROPERTY

END_INTERFACE

// ---- Components/Analog/Interface/I_AnalogChannel_Standard.TcIO
INTERFACE I_AnalogChannel_Standard EXTENDS I_AnalogChannel_Generic

PROPERTY Limit1High : BOOL
GET
END_GET
END_PROPERTY

PROPERTY Limit1Low : BOOL
GET
END_GET
END_PROPERTY

PROPERTY Limit2High : BOOL
GET
END_GET
END_PROPERTY

PROPERTY Limit2Low : BOOL
GET
END_GET
END_PROPERTY

END_INTERFACE

// ---- Components/Analog/Interface/I_AnalogInput.TcIO
INTERFACE I_AnalogInput EXTENDS I_Component, I_ForcibleInt

{attribute 'monitoring' := 'call'}
PROPERTY RawValue : INT
GET
END_GET
END_PROPERTY

{attribute 'monitoring' := 'call'}
PROPERTY Value : LREAL
GET
END_GET
END_PROPERTY

END_INTERFACE

// ---- Components/Analog/Interface/I_AnalogOutput.TcIO
INTERFACE I_AnalogOutput EXTENDS I_Component, I_ForcibleInt

{attribute 'monitoring' := 'call'}
PROPERTY RawValue : INT
GET
END_GET
SET
END_SET
END_PROPERTY

{attribute 'monitoring' := 'call'}
PROPERTY Value : LREAL
GET
END_GET
SET
END_SET
END_PROPERTY

END_INTERFACE

// ---- Components/CoE/Interface/I_CoeAccess.TcIO
INTERFACE I_CoeAccess EXTENDS I_Base

PROPERTY CoE : I_CoeDevice
GET
END_GET
END_PROPERTY

END_INTERFACE

// ---- Components/CoE/Interface/I_CoeDevice.TcIO
INTERFACE I_CoeDevice EXTENDS I_Component, I_TaskResult

PROPERTY AdsAddr : REFERENCE TO AMSADDR
GET
END_GET
SET
END_SET
END_PROPERTY

METHOD Read
VAR_INPUT
	Index	 : WORD;
	SubIndex : BYTE;
	pDstBuf	 : PVOID;
	BufLen	 : UDINT;
END_VAR
END_METHOD

METHOD Write
VAR_INPUT
	Index	 : WORD;
	SubIndex : BYTE;
	pDstBuf	 : PVOID;
	BufLen	 : UDINT;
END_VAR
END_METHOD

END_INTERFACE

// ---- Components/CoE/Interface/I_CoeTransfer.TcIO
// A CoE transfer that an I_CoeTransferScheduler services each cycle while Busy is TRUE.
INTERFACE I_CoeTransfer EXTENDS I_Cyclic, I_TaskResult

END_INTERFACE

// ---- Components/CoE/Interface/I_CoeTransferScheduler.TcIO
// Services registered CoE transfers each cycle until they report Busy = FALSE.
// EtherCatMaster implements it so that only transfers in flight cost cycle time.
INTERFACE I_CoeTransferScheduler EXTENDS I_Base

// Adds Transfer to the set serviced each cycle (idempotent). Returns FALSE if the set is full.
METHOD Register : BOOL
VAR_INPUT
	Transfer : I_CoeTransfer;
END_VAR
END_METHOD

END_INTERFACE

// ---- Components/Cylinder/Interface/I_Cylinder.TcIO
INTERFACE I_Cylinder EXTENDS I_CylinderCommand, I_CylinderStatus, I_Component, I_TaskResult, I_Resettable

{attribute 'monitoring' := 'call'}
PROPERTY ExtendTimeout : TIME
GET
END_GET
SET
END_SET
END_PROPERTY

{attribute 'monitoring' := 'call'}
PROPERTY RetractTimeout : TIME
GET
END_GET
SET
END_SET
END_PROPERTY

END_INTERFACE

// ---- Components/Cylinder/Interface/I_CylinderCommand.TcIO
INTERFACE I_CylinderCommand EXTENDS I_Base

METHOD Extend
END_METHOD

METHOD Retract
END_METHOD

END_INTERFACE

// ---- Components/Cylinder/Interface/I_CylinderStatus.TcIO
INTERFACE I_CylinderStatus EXTENDS I_Base

{attribute 'monitoring' := 'call'}
PROPERTY Extended : BOOL
GET
END_GET
END_PROPERTY

{attribute 'monitoring' := 'call'}
PROPERTY Extending : BOOL
GET
END_GET
END_PROPERTY

{attribute 'monitoring' := 'call'}
PROPERTY Retracted : BOOL
GET
END_GET
END_PROPERTY

{attribute 'monitoring' := 'call'}
PROPERTY Retracting : BOOL
GET
END_GET
END_PROPERTY

END_INTERFACE

// ---- Components/Digital/Interface/I_DigitalInput.TcIO
INTERFACE I_DigitalInput EXTENDS I_Component, I_ForcibleBool

{attribute 'monitoring' := 'call'}
PROPERTY IsActive : BOOL
GET
END_GET
END_PROPERTY

END_INTERFACE

// ---- Components/Digital/Interface/I_DigitalOutput.TcIO
INTERFACE I_DigitalOutput EXTENDS I_Component, I_ForcibleBool

{attribute 'monitoring' := 'call'}
PROPERTY On : BOOL
GET
END_GET
SET
END_SET
END_PROPERTY

END_INTERFACE

// ---- Components/EtherCat/Interface/I_EcIoDevice.TcIO
// One EtherCAT slave: decoded ESM / link flags, CoE access and the raw Tc2_EtherCAT
// configuration and extended state references.
INTERFACE I_EcIoDevice EXTENDS I_IoDevice, I_CoeAccess

{attribute 'monitoring' := 'call'}
PROPERTY Bootstrap : BOOL
GET
END_GET
END_PROPERTY

// Slave configuration data (address, mailbox sizes, ...) as read by FB_EcGetConfSlaves.
PROPERTY Configuration : REFERENCE TO ST_EcSlaveConfigData
GET
END_GET
END_PROPERTY

{attribute 'monitoring' := 'call'}
PROPERTY DeviceError : BOOL
GET
END_GET
END_PROPERTY

{attribute 'monitoring' := 'call'}
PROPERTY Disabled : BOOL
GET
END_GET
END_PROPERTY

{attribute 'monitoring' := 'call'}
PROPERTY Init : BOOL
GET
END_GET
END_PROPERTY

{attribute 'monitoring' := 'call'}
PROPERTY InitCmdError : BOOL
GET
END_GET
END_PROPERTY

{attribute 'monitoring' := 'call'}
PROPERTY InvalidVPRS : BOOL
GET
END_GET
END_PROPERTY

{attribute 'monitoring' := 'call'}
PROPERTY OP : BOOL
GET
END_GET
END_PROPERTY

{attribute 'monitoring' := 'call'}
PROPERTY PreOp : BOOL
GET
END_GET
END_PROPERTY

{attribute 'monitoring' := 'call'}
PROPERTY SafeOp : BOOL
GET
END_GET
END_PROPERTY

// Live extended slave state as read by FB_EcGetAllExtSlaveStates.
PROPERTY State : REFERENCE TO ST_EcExtendedSlaveState
GET
END_GET
END_PROPERTY

END_INTERFACE

// ---- Components/EtherCat/Interface/I_EcSlaveRegistry.TcIO
// Read-only view of the configured EtherCAT slaves, indexed 0-based in configuration order.
// EtherCatMaster implements it; SyncUnitTask and other collaborators that only need to resolve
// slaves depend on this contract instead of on the whole master.
INTERFACE I_EcSlaveRegistry EXTENDS I_Base

{attribute 'monitoring' := 'call'}
PROPERTY ConfiguredSlaveCount : UINT
GET
END_GET
END_PROPERTY

// Configured slave index (0-based) of the slave with EtherCAT address Addr, -1 if none.
// O(1) for the dense address range starting at 1001, linear search otherwise.
METHOD GetSlaveIndexByAddr : DINT
VAR_INPUT
	Addr : UINT;
END_VAR
END_METHOD

// Name of the configured slave at Index, '' if Index is out of range.
METHOD GetSlaveName : STRING
VAR_INPUT
	Index : UINT;
END_VAR
END_METHOD

// TRUE if the configured slave at Index belongs to a hot connect group (topology status bits 4 or 5).
// FALSE if Index is out of range.
METHOD IsHotConnectMember : BOOL
VAR_INPUT
	Index : UINT;
END_VAR
END_METHOD

END_INTERFACE

// ---- Components/EtherCat/Interface/I_EtherCatDiagnosticEventProvider.TcIO
INTERFACE I_EtherCatDiagnosticEventProvider EXTENDS I_EventReactionTcEvents

METHOD RaiseEtherCatDiagnosticEvent
VAR_INPUT
	EventId	  : UDINT;
	Argument1 : STRING := '';
	Argument2 : STRING := '';
	Argument3 : STRING := '';
END_VAR
END_METHOD

METHOD RaiseSyncUnitEvent
VAR_INPUT
	EventId	  : UDINT;
	Argument1 : STRING := '';
	Argument2 : STRING := '';
	Argument3 : STRING := '';
END_VAR
END_METHOD

END_INTERFACE

// ---- Components/EtherCat/Interface/I_EtherCatMasterDiagnostic.TcIO
// The slave registry members (ConfiguredSlaveCount, GetSlaveIndexByAddr, GetSlaveName, IsHotConnectMember)
// are inherited from I_EcSlaveRegistry.
INTERFACE I_EtherCatMasterDiagnostic EXTENDS I_Component, I_Resettable, I_EcSlaveRegistry

// Which subsystem produced ErrorId (see E_EcErrorSource for the meaning of ErrorId per source).
{attribute 'monitoring' := 'call'}
PROPERTY ErrorSource : E_EcErrorSource
GET
END_GET
END_PROPERTY

METHOD GetIoDeviceByAddr : I_EcIoDevice
VAR_INPUT
	Addr : WORD;
END_VAR
END_METHOD

METHOD GetIoDeviceByName : I_EcIoDevice
VAR_INPUT
	Name : STRING(31);
END_VAR
END_METHOD

{attribute 'monitoring' := 'call'}
PROPERTY LocalAmsNetId : T_AmsNetId
GET
END_GET
END_PROPERTY

{attribute 'monitoring' := 'call'}
PROPERTY MasterAmsNetId : T_AmsNetId
GET
END_GET
END_PROPERTY

METHOD RegisterEventProvider
VAR_INPUT
	EventProvider : I_EtherCatDiagnosticEventProvider;
END_VAR
END_METHOD

{attribute 'monitoring' := 'call'}
PROPERTY SlaveCount : UINT
GET
END_GET
END_PROPERTY

END_INTERFACE

// ---- Components/EtherCat/Interface/I_IoDevice.TcIO
INTERFACE I_IoDevice EXTENDS I_Base

{attribute 'monitoring' := 'call'}
PROPERTY IoDataValid : BOOL
GET
END_GET
END_PROPERTY

END_INTERFACE

// ---- Components/EtherCat/Interface/I_SyncUnitTask.TcIO
INTERFACE I_SyncUnitTask EXTENDS I_Component

{attribute 'monitoring' := 'call'}
PROPERTY IoDataValid : BOOL
GET
END_GET
END_PROPERTY

{attribute 'monitoring' := 'call'}
PROPERTY IsHotConnect : BOOL
GET
END_GET
END_PROPERTY

{attribute 'monitoring' := 'call'}
PROPERTY PUBLIC SlaveCount : UINT
GET
END_GET
END_PROPERTY

END_INTERFACE

// ---- Components/Recipe/Interface/I_RecipeManagment.TcIO
INTERFACE I_RecipeManagment EXTENDS I_Component

{attribute 'monitoring' := 'call'}
PROPERTY AutoLoadChangesToActive : BOOL
SET
END_SET
END_PROPERTY

{attribute 'monitoring' := 'call'}
PROPERTY ChangesPending : BOOL
GET
END_GET
END_PROPERTY

METHOD LoadChangesToActive
VAR_INPUT
END_VAR
END_METHOD

END_INTERFACE

// ---- Components/Safety/Interface/I_InSafetyGroup.TcIO
INTERFACE I_InSafetyGroup EXTENDS I_Base

PROPERTY SafetyGroup : I_TaskResult
SET
END_SET
END_PROPERTY

END_INTERFACE

// ---- Components/Safety/Interface/I_SafetyBase.TcIO
INTERFACE I_SafetyBase EXTENDS I_Component, I_Resettable, I_SafetySimulation, I_TaskResult

{attribute 'monitoring' := 'call'}
PROPERTY OK : BOOL
GET
END_GET
END_PROPERTY

PROPERTY ResetFunction : I_SafetyReset
SET
END_SET
END_PROPERTY

END_INTERFACE

// ---- Components/Safety/Interface/I_SafetyModule.TcIO
INTERFACE I_SafetyModule EXTENDS I_SafetySimulation, I_TaskResult, I_Resettable, I_Module

METHOD AddSafetyComponent
VAR_INPUT
	Component : I_SafetyBase;
END_VAR
END_METHOD

{attribute 'monitoring' := 'call'}
PROPERTY OK : BOOL
GET
END_GET
END_PROPERTY

PROPERTY SafetyPlcCoE : I_CoeDevice
GET
END_GET
END_PROPERTY

END_INTERFACE

// ---- Components/Safety/Interface/I_SafetyReset.TcIO
INTERFACE I_SafetyReset EXTENDS I_Cyclic, I_TaskResult

METHOD Execute
VAR_INPUT
END_VAR
END_METHOD

PROPERTY PulseDuration : TIME
SET
END_SET
END_PROPERTY

END_INTERFACE

// ---- Components/Safety/Interface/I_SafetySimulation.TcIO
INTERFACE I_SafetySimulation EXTENDS I_Simulatable

METHOD SimulateSafetyDiag
VAR_INPUT
	SimulationValueDiag : UINT;
END_VAR
END_METHOD

METHOD SimulateSafetyState
VAR_INPUT
	SimulationValueState : USINT;
END_VAR
END_METHOD

END_INTERFACE

// ---- Components/Serial/Interface/I_SerialByteConnection.TcIO
INTERFACE I_SerialByteConnection

PROPERTY ByteData : BYTE
GET
END_GET
END_PROPERTY

PROPERTY ByteDataRecieved : BOOL
GET
END_GET
END_PROPERTY

METHOD SendAByte : HRESULT
VAR_INPUT
	DataToSend : BYTE;
END_VAR
END_METHOD

END_INTERFACE

// ---- Components/Serial/Interface/I_SerialLineControl.TcIO
INTERFACE I_SerialLineControl EXTENDS I_Cyclic

PROPERTY rxBuffer : REFERENCE TO combuffer
GET
END_GET
END_PROPERTY

PROPERTY txBuffer : REFERENCE TO combuffer
GET
END_GET
END_PROPERTY

END_INTERFACE

// ---- Components/Serial/Interface/I_SerialStringConnection.TcIO
INTERFACE I_SerialStringConnection

METHOD SendAString : HRESULT
VAR_INPUT
	DataToSend : T_MaxString;
END_VAR
END_METHOD

PROPERTY StringData : t_maxstring
GET
END_GET
END_PROPERTY

PROPERTY StringRecieved : BOOL
GET
END_GET
END_PROPERTY

END_INTERFACE

// ---- Components/Tcp Ip/Interface/I_TcpIpConnection.TcIO
INTERFACE I_TcpIpConnection EXTENDS I_Component

{attribute 'monitoring' := 'call'}
PROPERTY ConnectionState : E_SocketConnectionState
GET
END_GET
END_PROPERTY

{attribute 'monitoring' := 'call'}
PROPERTY IP : T_IPv4Addr
SET
END_SET
END_PROPERTY

{attribute 'monitoring' := 'call'}
PROPERTY Port : UDINT
SET
END_SET
END_PROPERTY

METHOD RegisterCommand
VAR_INPUT
	Command : I_TcpIpSubscription;
END_VAR
END_METHOD

METHOD SendCommand
VAR_INPUT
	Command : POINTER TO ST_TcpIpPayload;
END_VAR
END_METHOD

METHOD SendPriorityCommand
VAR_INPUT
	Command : POINTER TO ST_TcpIpPayload;
END_VAR
END_METHOD

PROPERTY Socket : T_HSOCKET
GET
END_GET
END_PROPERTY

END_INTERFACE

// ---- Components/Tcp Ip/Interface/I_TcpIpSubscription.TcIO
INTERFACE I_TcpIpSubscription EXTENDS I_Base

METHOD UpdateCommandResult
VAR_INPUT
	Response : POINTER TO ST_TcpIpPayload;
END_VAR
END_METHOD

END_INTERFACE

// ---- Component/Interface/I_Component.TcIO
INTERFACE I_Component EXTENDS I_Base

METHOD Accept
VAR_INPUT
	ComponentVisitor : I_ComponentVisitor;
END_VAR
END_METHOD

METHOD DeregisterWithParent
VAR_INPUT
	Parent : I_ContainComponents;
END_VAR
END_METHOD

{attribute 'monitoring' := 'call'}
PROPERTY Name : T_MaxString
GET
END_GET
SET
END_SET
END_PROPERTY

METHOD RegisterWithParent
VAR_INPUT
	Parent : I_ContainComponents;
END_VAR
END_METHOD

END_INTERFACE

// ---- Component/Interface/I_ComponentVisitor.TcIO
INTERFACE I_ComponentVisitor

METHOD VisitComponent
VAR_INPUT
	Component : I_Component;
END_VAR
END_METHOD

END_INTERFACE

// ---- Events/Interface/I_EventArguments.TcIO
INTERFACE I_EventArguments EXTENDS I_Base

METHOD AddString : I_EventArguments
VAR_INPUT
	Argument : STRING;
END_VAR
END_METHOD

METHOD Clear : I_EventArguments
VAR_INPUT
END_VAR
END_METHOD

END_INTERFACE

// ---- Events/Interface/I_EventClass.TcIO
INTERFACE I_EventClass EXTENDS I_EventReaction, I_Resettable

METHOD PUBLIC Arguments : I_EventArguments
VAR_INPUT
	EventId : UDINT;
END_VAR
END_METHOD

METHOD PUBLIC ClearEventById
VAR_INPUT
	EventId : UDINT;
END_VAR
END_METHOD

{attribute 'monitoring' := 'call'}
PROPERTY IsResettable : BOOL
GET
END_GET
END_PROPERTY

METHOD PUBLIC RaiseEvent
VAR_INPUT
	EventId	  : UDINT;
END_VAR
END_METHOD

METHOD ResetBySeverity : BOOL
VAR_INPUT
	Severity : UDINT;
END_VAR
END_METHOD

METHOD SetEvent
VAR_INPUT
	EventId	  : UDINT;
	Trigger	  : POINTER TO BOOL;
	AutoReset : BOOL;
END_VAR
END_METHOD

END_INTERFACE

// ---- Events/Interface/I_EventClassTcEvents.TcIO
INTERFACE I_EventClassTcEvents EXTENDS I_EventClass

METHOD PUBLIC GenerateTcEvents
VAR_INPUT
	Name   : T_MaxString;
	pClass : PVOID; // ADR(TC_Events.XY) - TC Event Class in TypeSystem
	nSize  : UDINT; // SIZEOF(ST_XY) - TC Event Class in TypeSystem
END_VAR
END_METHOD

METHOD GetHighestActiveEventSeverity : TcEventSeverity
END_METHOD

END_INTERFACE

// ---- Events/Interface/I_EventReaction.TcIO
INTERFACE I_EventReaction EXTENDS I_Resettable

METHOD GetHighestActiveEventReaction : DINT;
END_METHOD

METHOD SetEventReactions
VAR_INPUT
	Verbose	 : DINT := 0;
	Info	 : DINT := 1;
	Warning	 : DINT := 2;
	Error	 : DINT := 3;
	Critical : DINT := 4;
END_VAR
END_METHOD

END_INTERFACE

// ---- Events/Interface/I_EventReactionTcEvents.TcIO
INTERFACE I_EventReactionTcEvents EXTENDS I_EventReaction

METHOD GetHighestActiveEventSeverity : TcEventSeverity
END_METHOD

END_INTERFACE

// ---- HMI/Interface/I_Button.TcIO
INTERFACE I_Button EXTENDS I_Base

{attribute 'monitoring' := 'call'}
PROPERTY Active : BOOL
GET
END_GET
END_PROPERTY

{attribute 'monitoring' := 'call'}
PROPERTY Name : STRING
GET
END_GET
SET
END_SET
END_PROPERTY

PROPERTY Permissive : I_Permissive
GET
END_GET
END_PROPERTY

END_INTERFACE

// ---- HMI/Interface/I_HmiFunction.TcIO
INTERFACE I_HmiFunction EXTENDS I_Component

{attribute 'monitoring' := 'call'}
PROPERTY ControlType : STRING
GET
END_GET
SET
END_SET
END_PROPERTY

METHOD Disable
VAR_INPUT
END_VAR
END_METHOD

METHOD Enable
VAR_INPUT
END_VAR
END_METHOD

{attribute 'monitoring' := 'call'}
PROPERTY Enabled : BOOL
GET
END_GET
END_PROPERTY

{attribute 'monitoring' := 'call'}
PROPERTY InstancePath : STRING
GET
END_GET
END_PROPERTY

{attribute 'monitoring' := 'call'}
PROPERTY LinkObject : STRING
GET
END_GET
SET
END_SET
END_PROPERTY

END_INTERFACE

// ---- HMI/Interface/I_Permissive.TcIO
INTERFACE I_Permissive EXTENDS I_Base

{attribute 'monitoring' := 'call'}
PROPERTY OK : BOOL
GET
END_GET
END_PROPERTY

METHOD Set
VAR_INPUT
	Index  : UDINT(0..9);
	Reason : STRING;
	Value  : BOOL;
END_VAR
END_METHOD

END_INTERFACE

// ---- HMI/Interface/I_StringCollection.TcIO
INTERFACE I_StringCollection

METHOD AddString
VAR_INPUT
	StringToAdd : T_MaxString;
END_VAR
END_METHOD

METHOD Clear : BOOL
VAR_INPUT
END_VAR
END_METHOD

PROPERTY Entries : UDINT
GET
END_GET
END_PROPERTY

END_INTERFACE

// ---- Kinematic Group/Interface/I_KinematicGroup.TcIO
INTERFACE I_KinematicGroup EXTENDS I_Component, I_Override, I_TaskResult, I_Resettable

METHOD AddAcsAxis : BOOL
VAR_INPUT
	AxisId : UDINT;
END_VAR
END_METHOD

METHOD AddMcsAxis : BOOL
VAR_INPUT
	AxisId : UDINT;
END_VAR
END_METHOD

METHOD BuildGroup
VAR_INPUT
END_VAR
END_METHOD

METHOD DissolveGroup
VAR_INPUT
END_VAR
END_METHOD

{attribute 'monitoring' := 'call'}
PROPERTY Status : E_KinStatus
GET
END_GET
END_PROPERTY

END_INTERFACE

// ---- Modes/Interface/I_Mode.TcIO
INTERFACE I_Mode EXTENDS I_Base

METHOD ChangeMode
VAR_INPUT
	RequestedMode : DINT;
END_VAR
END_METHOD

{attribute 'monitoring' := 'call'}
PROPERTY CurrentMode : DINT
GET
END_GET
END_PROPERTY

END_INTERFACE

// ---- Module/Interface/I_Module.TcIO
INTERFACE I_Module EXTENDS I_ContainComponents, I_ContainModules, I_Base

METHOD Accept
VAR_INPUT
	Visitor : I_ModuleVisitor;
END_VAR
END_METHOD

METHOD DeregisterWithParent
VAR_INPUT
	Parent : I_ContainModules;
END_VAR
END_METHOD

{attribute 'monitoring' := 'call'}
PROPERTY Name : T_MaxString
GET
END_GET
END_PROPERTY

METHOD RegisterWithParent
VAR_INPUT
	Parent : I_ContainModules;
END_VAR
END_METHOD

METHOD ResetComponents : BOOL
END_METHOD

METHOD ResetModules : BOOL
END_METHOD

END_INTERFACE

// ---- Module/Interface/I_ModuleVisitor.TcIO
INTERFACE I_ModuleVisitor

METHOD VisitModule
VAR_INPUT
	Module : I_Module;
END_VAR
END_METHOD

END_INTERFACE

// ---- Motion/Interface/I_AxisDynamics.TcIO
INTERFACE I_AxisDynamics EXTENDS I_Base

{attribute 'monitoring' := 'call'}
PROPERTY Acceleration : LREAL
GET
END_GET
SET
END_SET
END_PROPERTY

{attribute 'monitoring' := 'call'}
PROPERTY Deceleration : LREAL
GET
END_GET
SET
END_SET
END_PROPERTY

{attribute 'monitoring' := 'call'}
PROPERTY Jerk : LREAL
GET
END_GET
SET
END_SET
END_PROPERTY

{attribute 'monitoring' := 'call'}
PROPERTY Velocity : LREAL
GET
END_GET
SET
END_SET
END_PROPERTY

END_INTERFACE

// ---- Motion/Interface/I_AxisEnable.TcIO
INTERFACE I_AxisEnable EXTENDS I_Enablable

{attribute 'monitoring' := 'call'}
PROPERTY InhibitFeedBackward : BOOL
GET
END_GET
SET
END_SET
END_PROPERTY

{attribute 'monitoring' := 'call'}
PROPERTY InhibitFeedForward : BOOL
GET
END_GET
SET
END_SET
END_PROPERTY

END_INTERFACE

// ---- Motion/Interface/I_AxisHome.TcIO
INTERFACE I_AxisHome EXTENDS I_Base

METHOD Home
VAR_INPUT
END_VAR
END_METHOD

END_INTERFACE

// ---- Motion/Interface/I_AxisJog.TcIO
INTERFACE I_AxisJog EXTENDS I_Base

METHOD Jog
VAR_INPUT
	JogForward	 : BOOL;
	JogBackwards : BOOL;
	Distance	 : LREAL := 0;
END_VAR
END_METHOD

END_INTERFACE

// ---- Motion/Interface/I_AxisMoveAbsolute.TcIO
INTERFACE I_AxisMoveAbsolute EXTENDS I_Base

METHOD MoveAbsolute : BOOL
VAR_INPUT
	TargetPosition : LREAL;
	AbortPrevious  : BOOL := TRUE;
END_VAR
END_METHOD

END_INTERFACE

// ---- Motion/Interface/I_AxisMoveModulo.TcIO
INTERFACE I_AxisMoveModulo EXTENDS I_Base

METHOD MoveModulo : BOOL
VAR_INPUT
	Position	  : LREAL;
	AbortPrevious : BOOL		 := TRUE;
END_VAR
END_METHOD

END_INTERFACE

// ---- Motion/Interface/I_AxisMoveRelative.TcIO
INTERFACE I_AxisMoveRelative EXTENDS I_Base

METHOD MoveRelative : BOOL
VAR_INPUT
	Distance	  : LREAL;
	AbortPrevious : BOOL := TRUE;
END_VAR
END_METHOD

END_INTERFACE

// ---- Motion/Interface/I_AxisMoveVelocity.TcIO
INTERFACE I_AxisMoveVelocity EXTENDS I_Base

METHOD MoveVelocity : BOOL
VAR_INPUT
	Velocity	  : LREAL;
	AbortPrevious : BOOL := TRUE;
END_VAR
END_METHOD

END_INTERFACE

// ---- Motion/Interface/I_AxisStatus.TcIO
INTERFACE I_AxisStatus EXTENDS I_Base, I_TaskResult

{attribute 'monitoring' := 'call'}
PROPERTY ActualAcceleration : LREAL
GET
END_GET
END_PROPERTY

{attribute 'monitoring' := 'call'}
PROPERTY ActualPosition : LREAL
GET
END_GET
END_PROPERTY

{attribute 'monitoring' := 'call'}
PROPERTY ActualPositionModulo : LREAL
GET
END_GET
END_PROPERTY

{attribute 'monitoring' := 'call'}
PROPERTY ActualTorque : LREAL
GET
END_GET
END_PROPERTY

{attribute 'monitoring' := 'call'}
PROPERTY ActualVelocity : LREAL
GET
END_GET
END_PROPERTY

{attribute 'monitoring' := 'call'}
PROPERTY Coupled : BOOL
GET
END_GET
END_PROPERTY

{attribute 'monitoring' := 'call'}
PROPERTY Disabled : BOOL
GET
END_GET
END_PROPERTY

{attribute 'monitoring' := 'call'}
PROPERTY Enabled : BOOL
GET
END_GET
END_PROPERTY

{attribute 'monitoring' := 'call'}
PROPERTY PositionLag : LREAL
GET
END_GET
END_PROPERTY

{attribute 'monitoring' := 'call'}
PROPERTY SetAcceleration : LREAL
GET
END_GET
END_PROPERTY

{attribute 'monitoring' := 'call'}
PROPERTY SetPosition : LREAL
GET
END_GET
END_PROPERTY

{attribute 'monitoring' := 'call'}
PROPERTY SetPositionModulo : LREAL
GET
END_GET
END_PROPERTY

{attribute 'monitoring' := 'call'}
PROPERTY SetVelocity : LREAL
GET
END_GET
END_PROPERTY

{attribute 'monitoring' := 'call'}
PROPERTY SynchronizedMotion : BOOL
GET
END_GET
END_PROPERTY

{attribute 'monitoring' := 'call'}
PROPERTY Stopped : BOOL
GET
END_GET
END_PROPERTY

END_INTERFACE

// ---- Motion/Interface/I_Axis.TcIO
(* Motion generation independent view on an axis.
   Deliberately free of any Tc2_MC2 / Tc3_Mc3Ptp type so that generic consumers
   (HMI, event reactions, diagnostics) work against MC2 and MC3 alike.
   The raw AXIS_REF is NOT part of this abstraction. It is available one level
   down, on I_Mc2Axis / I_Mc3Axis, for code that deliberately targets one
   motion generation and needs direct access to the NC structure. *)
INTERFACE I_Axis EXTENDS I_Component, I_AxisEnable, I_Resettable, I_Stoppable, I_AxisDynamics, I_AxisStatus, I_AxisJog, I_AxisHome, I_AxisSettings, I_Override

{attribute 'monitoring' := 'call'}
PROPERTY ErrorId : UDINT
GET
END_GET
END_PROPERTY

PROPERTY MotionTasks : I_MotionTaskCollection
GET
END_GET
END_PROPERTY

END_INTERFACE

// ---- Motion/Interface/I_AxisGear.TcIO
(* Electronic gearing as an optional capability rather than an axis subtype.

   An axis that can be coupled to a master implements this in addition to
   I_Axis_PTP. Consumers discover it instead of assuming it:

       IF __QUERYINTERFACE(MyAxis, Gearing) THEN
           Gearing.GearOut();
       END_IF

   Whether an axis is currently coupled is reported by I_AxisStatus.Coupled,
   which is the NC's own view and is available on every axis. *)
INTERFACE I_AxisGear EXTENDS I_Base

(* Couples the slave to its configured master. *)
METHOD GearIn
VAR_INPUT
END_VAR
END_METHOD

(* Decouples the slave from its master. *)
METHOD GearOut
VAR_INPUT
END_VAR
END_METHOD

END_INTERFACE

// ---- Motion/Interface/I_AxisSettings.TcIO
(* Axis settings that are independent of the motion generation (MC2 / MC3).
   Generation specific settings live on I_Mc2Settings / I_Mc3Settings. *)
INTERFACE I_AxisSettings EXTENDS I_Base

{attribute 'monitoring' := 'call'}
PROPERTY JogMode : E_AxisJogMode
GET
END_GET
SET
END_SET
END_PROPERTY

END_INTERFACE

// ---- Motion/Interface/I_Axis_PTP.TcIO
(* Motion generation independent view on a point to point axis.
   Implemented by Mc2AxisPTP and Mc3AxisPTP. *)
INTERFACE I_Axis_PTP EXTENDS I_Axis, I_AxisMoveAbsolute, I_AxisMoveModulo, I_AxisMoveRelative, I_AxisMoveVelocity

END_INTERFACE

// ---- Motion/Interface/I_MotionTaskCollection.TcIO
(* Read only view on a motion task collection, independent of the motion
   generation. Adding and removing tasks is generation specific and stays on
   I_Mc2MotionTaskCollection / I_Mc3MotionTaskCollection. *)
INTERFACE I_MotionTaskCollection EXTENDS I_TaskResult

{attribute 'monitoring' := 'call'}
PROPERTY ErrorTask : T_MaxString
GET
END_GET
END_PROPERTY

END_INTERFACE

// ---- Motion/MC2/Interface/I_Mc2Axis.TcIO
(* MC2 flavour of I_Axis: everything generic, plus the MC2 specific settings
   and the raw Tc2_MC2.AXIS_REF via I_Mc2AxisRef.
   This interface is MC2 bound by design. Code that should work with MC2 and
   MC3 alike must be typed on I_Axis / I_Axis_PTP instead. *)
INTERFACE I_Mc2Axis EXTENDS I_Axis, I_Mc2Settings, I_Mc2AxisRef

END_INTERFACE

// ---- Motion/MC2/Interface/I_Mc2AxisGear.TcIO
INTERFACE I_Mc2AxisGear EXTENDS I_AxisGear

PROPERTY GearInMultiMasterOptions : ST_GearInMultiMasterOptions
SET
END_SET
END_PROPERTY

{attribute 'monitoring' := 'call'}
PROPERTY GearRatioMaster1 : LREAL
SET
END_SET
END_PROPERTY

{attribute 'monitoring' := 'call'}
PROPERTY GearRatioMaster2 : LREAL
SET
END_SET
END_PROPERTY

{attribute 'monitoring' := 'call'}
PROPERTY GearRatioMaster3 : LREAL
SET
END_SET
END_PROPERTY

{attribute 'monitoring' := 'call'}
PROPERTY GearRatioMaster4 : LREAL
SET
END_SET
END_PROPERTY

PROPERTY Master1 : I_Mc2Axis
SET
END_SET
END_PROPERTY

PROPERTY Master2 : I_Mc2Axis
SET
END_SET
END_PROPERTY

PROPERTY Master3 : I_Mc2Axis
SET
END_SET
END_PROPERTY

PROPERTY Master4 : I_Mc2Axis
SET
END_SET
END_PROPERTY

END_INTERFACE

// ---- Motion/MC2/Interface/I_Mc2Axis_PTP.TcIO
INTERFACE I_Mc2Axis_PTP EXTENDS I_Mc2Axis, I_Axis_PTP

END_INTERFACE

// ---- Motion/MC2/Interface/I_Mc2Settings.TcIO
(* MC2 specific settings. Generation independent settings (JogMode) live on
   I_AxisSettings so that generic consumers never touch a Tc2_MC2 type. *)
INTERFACE I_Mc2Settings EXTENDS I_Base

PROPERTY AxisParameterSet : REFERENCE TO ST_AxisParameterSet
GET
END_GET
END_PROPERTY

PROPERTY BufferMode : REFERENCE TO tc2_mc2.MC_BufferMode
GET
END_GET
END_PROPERTY

PROPERTY Direction : REFERENCE TO TC2_Mc2.MC_Direction
GET
END_GET
END_PROPERTY

PROPERTY MoveOptions : REFERENCE TO tc2_mc2.ST_MoveOptions
GET
END_GET
END_PROPERTY

END_INTERFACE

// ---- Motion/MC2/Interface/I_Mc2SlaveAxis.TcIO
INTERFACE I_Mc2SlaveAxis EXTENDS I_Mc2Axis_PTP, I_Mc2AxisGear

END_INTERFACE

// ---- Motion/MC3/Interface/I_Mc3SlaveAxis.TcIO
INTERFACE I_Mc3SlaveAxis EXTENDS I_Mc3Axis_PTP, I_Mc3AxisGear

END_INTERFACE

// ---- Motion/MC3/Interface/I_Mc3AxisGear.TcIO
INTERFACE I_Mc3AxisGear EXTENDS I_AxisGear

{attribute 'monitoring' := 'call'}
PROPERTY InGear : BOOL
GET
END_GET
END_PROPERTY

PROPERTY Master : I_Mc3Axis
SET
END_SET
END_PROPERTY

{attribute 'monitoring' := 'call'}
PROPERTY MasterHasError : BOOL
GET
END_GET
END_PROPERTY

{attribute 'monitoring' := 'call'}
PROPERTY RatioDenominator : UDINT
SET
END_SET
END_PROPERTY

{attribute 'monitoring' := 'call'}
PROPERTY RatioNumerator : UDINT
SET
END_SET
END_PROPERTY

PROPERTY ReactionToMasterError : EReactionToMasterError
SET
END_SET
END_PROPERTY

PROPERTY ReactionToSlaveError : EReactionToSlaveError
SET
END_SET
END_PROPERTY

END_INTERFACE

// ---- Motion/MC3/Interface/I_Mc3Axis_PTP.TcIO
INTERFACE I_Mc3Axis_PTP EXTENDS I_Mc3Axis, I_Axis_PTP

END_INTERFACE

// ---- Motion/MC3/Interface/I_Mc3Settings.TcIO
(* MC3 specific settings. Generation independent settings (JogMode) live on
   I_AxisSettings so that generic consumers never touch a Tc3_Mc3Ptp type. *)
INTERFACE I_Mc3Settings EXTENDS I_Base

PROPERTY BufferMode : REFERENCE TO Tc3_Mc3Ptp.EBufferMode
GET
END_GET
END_PROPERTY

PROPERTY Direction : REFERENCE TO Tc3_Mc3Ptp.EModuloDirection
GET
END_GET
END_PROPERTY

END_INTERFACE

// ---- Motion/MC3/Interface/I_Mc3Axis.TcIO
(* MC3 flavour of I_Axis: everything generic, plus the MC3 specific settings
   and the raw Tc3_Mc3Ptp.AXIS_REF via I_Mc3AxisRef.
   This interface is MC3 bound by design. Code that should work with MC2 and
   MC3 alike must be typed on I_Axis / I_Axis_PTP instead. *)
INTERFACE I_Mc3Axis EXTENDS I_Axis, I_Mc3Settings, I_Mc3AxisRef

END_INTERFACE

// ---- Statemachine/Interface/I_ContainStatemachine.TcIO
INTERFACE I_ContainStatemachine EXTENDS I_Base

PROPERTY Statemachine : I_Statemachine
GET
END_GET
END_PROPERTY

END_INTERFACE

// ---- Statemachine/Interface/I_State.TcIO
INTERFACE I_State EXTENDS I_Base

METHOD Executing : BOOL;
END_METHOD

METHOD Inactive
VAR_INPUT
END_VAR
END_METHOD

END_INTERFACE

// ---- Statemachine/Interface/I_Statemachine.TcIO
INTERFACE I_Statemachine EXTENDS I_Component

METHOD ChangeState
VAR_INPUT
	StateCommand : DINT;
END_VAR
END_METHOD

{attribute 'monitoring' := 'call'}
PROPERTY CurrentState : DINT
GET
END_GET
END_PROPERTY

PROPERTY Mode : I_Mode
GET
END_GET
SET
END_SET
END_PROPERTY

PROPERTY States : I_StateList
GET
END_GET
END_PROPERTY

END_INTERFACE

// ---- Utilities/AnyBuffer/Interface/I_AnyBuffer.TcIO
INTERFACE I_AnyBuffer

// Clears all buffer data and resets metadata to initial state
METHOD Clear : BOOL
END_METHOD

PROPERTY Configuration : REFERENCE TO ST_BufferConfiguration
GET
END_GET
END_PROPERTY

// Deletes element at specified index position and decrements element count
METHOD DeleteAtIndex : BOOL
VAR_INPUT
	index : DINT; // Zero-based index position of element to delete
END_VAR
END_METHOD

PROPERTY isEmpty : BOOL
GET
END_GET
END_PROPERTY

PROPERTY isFull : BOOL
GET
END_GET
END_PROPERTY

PROPERTY Metadata : REFERENCE TO ST_BufferMetadata
GET
END_GET
END_PROPERTY

// Retrieve an element at a specific index without removing it from the buffer
METHOD PeekAtIndex : BOOL
VAR_INPUT
	index	: DINT;
	element : ANY;
END_VAR
END_METHOD

// Remove and retrieve an element at a specific index, shifting remaining elements left
METHOD PopAtIndex : BOOL
VAR_INPUT
	index	   : DINT;
	element	   : ANY;
	popDiscard : BOOL := FALSE;
END_VAR
END_METHOD

// Removes and retrieves the first element from the buffer (FIFO/queue operation)
METHOD PopLeft : BOOL
VAR_INPUT
	element	   : ANY;			// Variable to receive the popped element
	popDiscard : BOOL := FALSE; // When TRUE, element is removed but not copied (type checking skipped)
END_VAR
END_METHOD

// Removes and retrieves the last element from the buffer (stack pop operation)
METHOD PopRight : BOOL
VAR_INPUT
	element	   : ANY;			// Variable to receive the popped element
	popDiscard : BOOL := FALSE; // When TRUE, element is removed but not copied (type checking skipped)
END_VAR
END_METHOD

// Add an element at a specific index, shifting remaining elements right
METHOD PushAtIndex : BOOL
VAR_INPUT
	index	: DINT;
	element : ANY;
END_VAR
END_METHOD

// Appends a new element to the left side of the buffer (LIFO/stack push operation)
METHOD PushLeft : BOOL
VAR_INPUT
	element : ANY;
END_VAR
END_METHOD

// Appends a new element to the right side of the buffer (FIFO/queue enqueue operation)
METHOD PushRight : BOOL
VAR_INPUT
	element : ANY;
END_VAR
END_METHOD

// Replaces an element at a specific index with the given element
METHOD ReplaceAtIndex : BOOL
VAR_INPUT
	index	: DINT;
	element : ANY;
END_VAR
END_METHOD

END_INTERFACE

// ---- Utilities/AnyBuffer/Interface/I_AnyBufferStrategy.TcIO
INTERFACE I_AnyBufferStrategy

METHOD Clear : BOOL
END_METHOD

PROPERTY isEmpty : BOOL
GET
END_GET
END_PROPERTY

PROPERTY isFull : BOOL
GET
END_GET
END_PROPERTY

END_INTERFACE

// ---- Utilities/File/Interface/I_FileHandler.TcIO
INTERFACE I_FileHandler EXTENDS I_Component, I_Cyclic, I_TaskResult, I_TaskResult, I_Resettable

METHOD ClearDocument
VAR_INPUT
END_VAR
END_METHOD

PROPERTY Datatype : T_MaxString
SET
END_SET
END_PROPERTY

METHOD LoadFile
END_METHOD

PROPERTY nData : UDINT
SET
END_SET
END_PROPERTY

PROPERTY PUBLIC Path : T_MaxString
GET
END_GET
SET
END_SET
END_PROPERTY

PROPERTY pData : PVOID
SET
END_SET
END_PROPERTY

METHOD ReadSymbol
END_METHOD

METHOD SaveFile
END_METHOD

PROPERTY SymbolName : T_MaxString
SET
END_SET
END_PROPERTY

PROPERTY Timeout : TIME
SET
END_SET
END_PROPERTY

METHOD UpdateSymbol
END_METHOD

END_INTERFACE

// ---- Utilities/Force/Interface/I_ForcibleBool.TcIO
INTERFACE I_ForcibleBool EXTENDS I_Base

{attribute 'monitoring' := 'call'}
PROPERTY Force : E_ForceState
GET
END_GET
SET
END_SET
END_PROPERTY

END_INTERFACE

// ---- Utilities/Force/Interface/I_ForcibleInt.TcIO
INTERFACE I_ForcibleInt

{attribute 'monitoring' := 'call'}
PROPERTY Force : E_ForceState
GET
END_GET
SET
END_SET
END_PROPERTY

PROPERTY ForceValue : INT
GET
END_GET
SET
END_SET
END_PROPERTY

END_INTERFACE

// ---- Utilities/Scaling/Interface/I_AnalogScalable.TcIO
INTERFACE I_AnalogScalable EXTENDS I_Base

PROPERTY Scale : I_AnalogScale
GET
END_GET
SET
END_SET
END_PROPERTY

END_INTERFACE

// ---- Utilities/Scaling/Interface/I_AnalogScale.TcIO
INTERFACE I_AnalogScale EXTENDS I_TransformLrealValue

PROPERTY InputMaximum : LREAL
GET
END_GET
SET
END_SET
END_PROPERTY

PROPERTY InputMinimum : LREAL
GET
END_GET
SET
END_SET
END_PROPERTY

PROPERTY OutputMaximum : LREAL
GET
END_GET
SET
END_SET
END_PROPERTY

PROPERTY OutputMinimum : LREAL
GET
END_GET
SET
END_SET
END_PROPERTY

END_INTERFACE

// ---- Utilities/Scaling/Interface/I_CalibratableLinear.TcIO
INTERFACE I_CalibratableLinear EXTENDS I_Base

PROPERTY CalibrateLinear : I_CalibrateLinear
GET
END_GET
SET
END_SET
END_PROPERTY

END_INTERFACE

// ---- Utilities/Scaling/Interface/I_CalibrateLinear.TcIO
INTERFACE I_CalibrateLinear EXTENDS I_TransformLrealValue

PROPERTY Gain : LREAL
SET
END_SET
END_PROPERTY

PROPERTY Offset : LREAL
SET
END_SET
END_PROPERTY

END_INTERFACE

// ---- Utilities/Scaling/Interface/I_TransformLRealValue.TcIO
INTERFACE I_TransformLRealValue EXTENDS I_Base

METHOD Transform : LREAL
VAR_INPUT
	Value	: LREAL;
	Reverse : BOOL := FALSE;
END_VAR
END_METHOD

END_INTERFACE

// ---- _Interface/I_Command.TcIO
INTERFACE I_Command EXTENDS I_Base

METHOD Execute : BOOL
VAR_INPUT
END_VAR
END_METHOD

END_INTERFACE

// ---- _Interface/I_Disposable.TcIO
INTERFACE I_Disposable EXTENDS I_Base

METHOD Dispose
VAR_INPUT
END_VAR
END_METHOD

END_INTERFACE

// ---- _Interface/I_Enablable.TcIO
INTERFACE I_Enablable EXTENDS I_Base

METHOD Disable
VAR_INPUT
END_VAR
END_METHOD

METHOD Enable
VAR_INPUT
END_VAR
END_METHOD

{attribute 'monitoring' := 'call'}
PROPERTY Enabled : BOOL
GET
END_GET
END_PROPERTY

END_INTERFACE

// ---- _Interface/I_Initializable.TcIO
INTERFACE I_Initializable EXTENDS I_Base

METHOD Initialize
END_METHOD

{attribute 'monitoring' := 'call'}
PROPERTY Initialized : BOOL
GET
END_GET
SET
END_SET
END_PROPERTY

END_INTERFACE

// ---- _Interface/I_Override.TcIO
INTERFACE I_Override EXTENDS I_Base

{attribute 'monitoring' := 'call'}
PROPERTY Override : LREAL
SET
END_SET
END_PROPERTY

END_INTERFACE

// ---- _Interface/I_Resettable.TcIO
INTERFACE I_Resettable EXTENDS I_Base

METHOD Reset
END_METHOD

END_INTERFACE

// ---- _Interface/I_Simulatable.TcIO
INTERFACE I_Simulatable EXTENDS I_Base

{attribute 'monitoring' := 'call'}
PROPERTY Simulated : BOOL
GET
END_GET
SET
END_SET
END_PROPERTY

END_INTERFACE

// ---- _Interface/I_Stoppable.TcIO
INTERFACE I_Stoppable EXTENDS I_Base

METHOD Stop
VAR_INPUT
END_VAR
END_METHOD

{attribute 'monitoring' := 'call'}
PROPERTY Stopped : BOOL
GET
END_GET
END_PROPERTY

END_INTERFACE

// ---- _Interface/I_TaskResult.TcIO
INTERFACE I_TaskResult EXTENDS I_Base

{attribute 'monitoring' := 'call'}
PROPERTY Busy : BOOL
GET
END_GET
END_PROPERTY

{attribute 'monitoring' := 'call'}
PROPERTY Error : BOOL
GET
END_GET
END_PROPERTY

{attribute 'monitoring' := 'call'}
PROPERTY ErrorId : UDINT
GET
END_GET
END_PROPERTY

END_INTERFACE

// ---- _Internal/CollectionPeeker/Interface/I_CollectionPeeker.TcIO
INTERFACE I_CollectionPeeker EXTENDS I_Base

{attribute 'monitoring':='call'}
PROPERTY CollectionName : T_MaxString
GET
END_GET
SET
END_SET
END_PROPERTY

{attribute 'monitoring':='call'}
PROPERTY FirstItem : UDINT
GET
END_GET
END_PROPERTY

{attribute 'monitoring':='call'}
PROPERTY LastItem : UDINT
GET
END_GET
END_PROPERTY

{attribute 'monitoring' := 'call'}
PROPERTY MoveDownOne : BOOL
SET
END_SET
END_PROPERTY

{attribute 'monitoring' := 'call'}
PROPERTY MoveUpOne : BOOL
SET
END_SET
END_PROPERTY

{attribute 'monitoring' := 'call'}
PROPERTY PageDown : BOOL
SET
END_SET
END_PROPERTY

{attribute 'monitoring' := 'call'}
PROPERTY PageUp : BOOL
SET
END_SET
END_PROPERTY

METHOD PeekAt
VAR_INPUT
	Peekable : I_Peekable;
END_VAR
END_METHOD

{attribute 'monitoring':='call'}
PROPERTY Refresh : BOOL
GET
END_GET
SET
END_SET
END_PROPERTY

END_INTERFACE

// ---- _Internal/CollectionPeeker/Interface/I_Peekable.TcIO
INTERFACE I_Peekable EXTENDS I_Base

METHOD AcceptPeeker
VAR_INPUT
	Peeker : I_Peeker;
END_VAR
END_METHOD

END_INTERFACE

// ---- _Internal/CollectionPeeker/Interface/I_Peeker.TcIO
INTERFACE I_Peeker EXTENDS I_Base

METHOD PeekCollection
VAR_INPUT
	Collection : I_Collection;
END_VAR
END_METHOD

END_INTERFACE

// ---- _Internal/Collection/Interface/I_Collection.TcIO
INTERFACE I_Collection EXTENDS I_Enumerator

METHOD AddItem
VAR_INPUT
	Item : I_Base;
END_VAR
END_METHOD

METHOD Clear
VAR_INPUT
END_VAR
END_METHOD

{attribute 'monitoring' := 'call'}
PROPERTY Count : UDINT
GET
END_GET
END_PROPERTY

{attribute 'monitoring' := 'call'}
PROPERTY IsEmpty : BOOL
GET
END_GET
END_PROPERTY

METHOD RemoveItem
VAR_INPUT
	Item : I_Base;
END_VAR
END_METHOD

END_INTERFACE

// ---- _Internal/Collection/Interface/I_Enumerator.TcIO
INTERFACE I_Enumerator

PROPERTY Current : I_Base
GET
END_GET
END_PROPERTY

{attribute 'monitoring' := 'call'}
PROPERTY CurrentItem : UDINT
GET
END_GET
END_PROPERTY

PROPERTY MoveToNext : BOOL
GET
END_GET
END_PROPERTY

METHOD ResetIterator
VAR_INPUT
END_VAR
END_METHOD

END_INTERFACE

// ---- _Internal/Component/Interface/I_ComponentCollection.TcIO
INTERFACE I_ComponentCollection EXTENDS I_Base

METHOD Accept
VAR_INPUT
	Visitor : I_ComponentVisitor;
END_VAR
END_METHOD

{attribute 'monitoring' := 'call'}
PROPERTY Count : UDINT
GET
END_GET
END_PROPERTY

METHOD GetAtIndex : I_Component
VAR_INPUT
	Index : UDINT;
END_VAR
END_METHOD

METHOD GetComponentByName : I_Component
VAR_INPUT
	Name : T_MaxString;
END_VAR
END_METHOD

END_INTERFACE

// ---- _Internal/Component/Interface/I_ContainComponents.TcIO
INTERFACE I_ContainComponents EXTENDS I_Base

PROPERTY Components : I_ComponentCollection
GET
END_GET
END_PROPERTY

METHOD DeregisterComponent  : RegistrationResult
VAR_INPUT
	Component : I_Component;
END_VAR
END_METHOD

METHOD DeregisterCyclic : RegistrationResult
VAR_INPUT
	Cyclic : I_Cyclic;
END_VAR
END_METHOD

METHOD DeregisterInitialize : RegistrationResult
VAR_INPUT
	Initializable : I_Initializable;
END_VAR
END_METHOD

METHOD RegisterComponent  : RegistrationResult
VAR_INPUT
	Component : I_Component;
END_VAR
END_METHOD

METHOD RegisterCyclic  : RegistrationResult
VAR_INPUT
	Cyclic : I_Cyclic;
END_VAR
END_METHOD

METHOD RegisterInitialize  : RegistrationResult
VAR_INPUT
	Initializable : I_Initializable;
END_VAR
END_METHOD

END_INTERFACE

// ---- _Internal/Cyclic/Interface/I_Cyclic.TcIO
INTERFACE I_Cyclic EXTENDS I_Base

METHOD CyclicLogic
VAR_INPUT
END_VAR
END_METHOD

END_INTERFACE

// ---- _Internal/List/Interface/I_List.TcIO
INTERFACE I_List EXTENDS I_Collection

METHOD ContainsItem : BOOL
VAR_INPUT
	Item : I_Base;
	;
END_VAR
END_METHOD

METHOD GetAtIndex : I_Base
VAR_INPUT
	Index : UDINT;
END_VAR
END_METHOD

METHOD InsertAtIndex : BOOL
VAR_INPUT
	Item  : I_Base;
	Index : UDINT;
END_VAR
END_METHOD

METHOD RemoveAtIndex
VAR_INPUT
	Index : UDINT;
END_VAR
END_METHOD

END_INTERFACE

// ---- _Internal/Module/Interface/I_ContainModules.TcIO
INTERFACE I_ContainModules EXTENDS I_Base

METHOD DeregisterCyclic : RegistrationResult
VAR_INPUT
	Cyclic : I_Cyclic;
END_VAR
END_METHOD

METHOD DeregisterInitialize : RegistrationResult
VAR_INPUT
	Initializable : I_Initializable;
END_VAR
END_METHOD

METHOD DeregisterModule : RegistrationResult
VAR_INPUT
	Module : I_Module;
END_VAR
END_METHOD

PROPERTY Modules : I_ModuleCollection
GET
END_GET
END_PROPERTY

METHOD RegisterCyclic  : RegistrationResult
VAR_INPUT
	Cyclic : I_Cyclic;
END_VAR
END_METHOD

METHOD RegisterInitialize  : RegistrationResult
VAR_INPUT
	Initializable : I_Initializable;
END_VAR
END_METHOD

METHOD RegisterModule  : RegistrationResult
VAR_INPUT
	Module : I_Module;
END_VAR
END_METHOD

END_INTERFACE

// ---- _Internal/Module/Interface/I_ModuleCollection.TcIO
INTERFACE I_ModuleCollection EXTENDS I_Base

METHOD Accept
VAR_INPUT
	Visitor : I_ModuleVisitor;
END_VAR
END_METHOD

{attribute 'monitoring' := 'call'}
PROPERTY Count : UDINT
GET
END_GET
END_PROPERTY

METHOD GetAtIndex : I_Module
VAR_INPUT
	Index : UDINT;
END_VAR
END_METHOD

METHOD GetModuleByName : I_Module
VAR_INPUT
	Name : T_MaxString;
END_VAR
END_METHOD

END_INTERFACE

// ---- _Internal/MotionTasks/MC2/Interface/I_Mc2AxisRef.TcIO
INTERFACE I_Mc2AxisRef

PROPERTY Axis : REFERENCE TO Tc2_MC2.AXIS_REF
GET
END_GET
END_PROPERTY

END_INTERFACE

// ---- _Internal/MotionTasks/MC2/Interface/I_Mc2MotionJogTask.TcIO
INTERFACE I_Mc2MotionJogTask EXTENDS I_Mc2MotionTask

PROPERTY JogBackwards : BOOL
SET
END_SET
END_PROPERTY

PROPERTY JogForward : BOOL
SET
END_SET
END_PROPERTY

PROPERTY Mode : E_JogMode
SET
END_SET
END_PROPERTY

PROPERTY Position : LREAL
SET
END_SET
END_PROPERTY

END_INTERFACE

// ---- _Internal/MotionTasks/MC2/Interface/I_Mc2MotionPowerTask.TcIO
INTERFACE I_Mc2MotionPowerTask EXTENDS I_Mc2MotionTask, I_AxisEnable

END_INTERFACE

// ---- _Internal/MotionTasks/MC2/Interface/I_Mc2MotionTask.TcIO
INTERFACE I_Mc2MotionTask EXTENDS I_Cyclic, I_TaskResult, I_Command

PROPERTY Axis : I_Mc2Axis
GET
END_GET
SET
END_SET
END_PROPERTY

{attribute 'monitoring' := 'call'}
PROPERTY Name : T_MaxString
GET
END_GET
SET
END_SET
END_PROPERTY

END_INTERFACE

// ---- _Internal/MotionTasks/MC2/Interface/I_Mc2MotionTaskCollection.TcIO
INTERFACE I_Mc2MotionTaskCollection EXTENDS I_MotionTaskCollection

METHOD AddTask
VAR_INPUT
	Task : I_Mc2MotionTask;
END_VAR
END_METHOD

METHOD RemoveTaskByInstance
VAR_INPUT
	Task : I_Mc2MotionTask;
END_VAR
END_METHOD

END_INTERFACE

// ---- _Internal/MotionTasks/MC3/Interface/I_Mc3AxisRef.TcIO
INTERFACE I_Mc3AxisRef

PROPERTY Axis : REFERENCE TO Tc3_Mc3Ptp.AXIS_REF
GET
END_GET
END_PROPERTY

END_INTERFACE

// ---- _Internal/MotionTasks/MC3/Interface/I_Mc3MotionJogTask.TcIO
INTERFACE I_Mc3MotionJogTask EXTENDS I_Mc3MotionTask

PROPERTY Distance : LREAL
SET
END_SET
END_PROPERTY

PROPERTY JogBackwards : BOOL
SET
END_SET
END_PROPERTY

PROPERTY JogForward : BOOL
SET
END_SET
END_PROPERTY

PROPERTY Mode : Tc3_Mc3Ptp.EJogMode
SET
END_SET
END_PROPERTY

END_INTERFACE

// ---- _Internal/MotionTasks/MC3/Interface/I_Mc3MotionPowerTask.TcIO
INTERFACE I_Mc3MotionPowerTask EXTENDS I_Mc3MotionTask, I_AxisEnable

END_INTERFACE

// ---- _Internal/MotionTasks/MC3/Interface/I_Mc3MotionTaskCollection.TcIO
INTERFACE I_Mc3MotionTaskCollection EXTENDS I_MotionTaskCollection

METHOD AddTask
VAR_INPUT
	Task : I_Mc3MotionTask;
END_VAR
END_METHOD

METHOD RemoveTaskByInstance
VAR_INPUT
	Task : I_Mc3MotionTask;
END_VAR
END_METHOD

END_INTERFACE

// ---- _Internal/MotionTasks/MC3/Interface/I_Mc3MotionTask.TcIO
INTERFACE I_Mc3MotionTask EXTENDS I_Cyclic, I_TaskResult, I_Command

PROPERTY Axis : I_Mc3Axis
GET
END_GET
SET
END_SET
END_PROPERTY

{attribute 'monitoring' := 'call'}
PROPERTY Name : T_MaxString
GET
END_GET
SET
END_SET
END_PROPERTY

END_INTERFACE

// ---- _Internal/Statemachine/Interface/I_StateList.TcIO
INTERFACE I_StateList

METHOD AddStateAtIndex
VAR_INPUT
	Index : DINT;
	State : I_State;
END_VAR
END_METHOD

METHOD GetStateAtIndex : I_State
VAR_INPUT
	Index : DINT;
END_VAR
END_METHOD

PROPERTY NumberOfStates : DINT
GET
END_GET
END_PROPERTY

END_INTERFACE

// ---- _Internal/Tracing/Interface/I_TraceArgument.TcIO
INTERFACE I_TraceArgument EXTENDS I_Base, I_ToString

END_INTERFACE

// ---- Components/EtherCat/EtherCatMaster.TcPOU
FUNCTION_BLOCK EtherCatMaster
VAR_GENERIC CONSTANT
	FRAMES	   : UINT := 1;
	SYNC_UNITS : UINT := 2;
END_VAR
EXTENDS CyclicComponent IMPLEMENTS I_EtherCatMasterDiagnostic, I_Initializable, I_TaskResult, I_Simulatable, I_CoeTransferScheduler
VAR
	EcMaster	AT %I*	: ST_EtherCatMasterInfo;
	FrmXWcState AT %I*	: ARRAY[0..(FRAMES - 1)] OF WORD;
	ConfiguredSlaveInfo : ARRAY[0..MAX_EC_SLAVES] OF ST_EcSlaveConfigData;
	SlavesState			: ARRAY[0..MAX_EC_SLAVES] OF ST_EcExtendedSlaveState;
	SlaveTopologyInfo	: ARRAY[0..MAX_EC_SLAVES] OF ST_TopologyDataEx;
	// Configured slave index + 1 by (EtherCAT address - FIRST_SLAVE_ADDR); 0 = no slave at that address
	AddrToIndex			: ARRAY[0..MAX_EC_SLAVES] OF UINT;
	// The sync units resolve their slaves through the I_EcSlaveRegistry role of this master
	SyncUnit			: ARRAY[0..(SYNC_UNITS - 1)] OF SyncUnitTask('Sync Unit', THIS^);
	IoDevice			: ARRAY[0..MAX_EC_SLAVES] OF EtherCatIoDevice('Io Device');
	// CoE transfers in flight - only these are serviced each cycle (I_CoeTransferScheduler)
	ActiveCoe			: ARRAY[0..MAX_EC_SLAVES] OF I_CoeTransfer;
	ActiveCoeCount		: UINT;
	EventProvider		: I_EtherCatDiagnosticEventProvider;
END_VAR

VAR
	InitSequenceState								 : UDINT;
	SlaveSequence									 : UDINT;
	RunSlaveDiag, LastFramesWcStatesOk				 : BOOL;
	LastChangeCount, LastSlaveCount, LastMasterState : UINT;
	EcStartupCycles									 : UINT;
	SlaveCountUsed									 : UINT;  // configured slaves covered by the arrays, latched in Initialize
	ScanIndex										 : UINT;  // slave position of the running multi-cycle pass
	SyncUnitScan									 : UINT;  // sync unit of the running assignment pass
	FirstDiagIndex									 : UINT;  // first slave that is not OP or reports a link problem
	AnyDiag											 : BOOL;
	SyncUnitsAssigned								 : BOOL;
	WaitCycles										 : UDINT; // ADS watchdog of the running wait step
	GetConfiguredSlaves								 : FB_EcGetConfSlaves;
	GetMasterFrameCount								 : FB_EcMasterFrameCount;
	GetAllSlaveStates								 : FB_EcGetAllExtSlaveStates;
	GetSlaveTopologyInfo							 : FB_EcGetSlaveTopologyInfo;
END_VAR

VAR
	{attribute 'hide'}
	_Initialized : BOOL;
	{attribute 'hide'}
	_Error : BOOL;
	{attribute 'hide'}
	_Busy : BOOL;
	{attribute 'hide'}
	_ErrorId : UDINT;
	{attribute 'hide'}
	_ErrorSource : E_EcErrorSource;
	{attribute 'hide'}
	_Simulated : BOOL;
	{attribute 'hide'}
	Config : ST_EcSlaveConfigData;
	{attribute 'hide'}
	State : ST_EcExtendedSlaveState;
	{attribute 'hide'}
	NullIoDevice : EtherCatIoDevice('NullIoDevice') := (Configuration := Config, State := State);
	{attribute 'hide'}
	_LocalAmsNetId : T_AmsNetId;
	{attribute 'hide'}
	_MasterAmsNetId : T_AmsNetId;
END_VAR

VAR CONSTANT
	FIRST_SLAVE_ADDR  : UINT  := 1001;	 // TwinCAT assigns EtherCAT addresses from 1001 in configuration order
	ADS_TIMEOUT		  : TIME  := T#5S;
	ERROR_ADS_TIMEOUT : UDINT := 16#745; // ADS client: timeout elapsed (watchdog abort)
END_VAR

// Counts the cycles of the running wait step; TRUE once MaxCycles is exceeded.
METHOD PRIVATE AdsWatchdogExpired : BOOL
VAR_INPUT
	MaxCycles : UDINT;
END_VAR
WaitCycles		   := WaitCycles + 1;
AdsWatchdogExpired := WaitCycles > MaxCycles;
END_METHOD

// Rebuilds the address map from the configured slaves (SlaveCountUsed entries).
METHOD PROTECTED BuildAddrToIndex
VAR
	i : UINT;
END_VAR
MEMSET(ADR(AddrToIndex), 0, SIZEOF(AddrToIndex));

i := 0;
WHILE i < SlaveCountUsed DO
	MapSlaveAddress(i);
	i := i + 1;
END_WHILE
END_METHOD

// TRUE while a diagnostic sequence runs. A pass over n slaves takes up to n / SLAVES_PER_CYCLE cycles,
// so Error/ErrorId of a change land that many cycles after the trigger.
{attribute 'monitoring' := 'call'}
PROPERTY Busy : BOOL
GET
Busy := _Busy;
END_GET
END_PROPERTY

{attribute 'monitoring' := 'call'}
PROPERTY ConfiguredSlaveCount : UINT
GET
ConfiguredSlaveCount := EcMaster.CfgSlaveCount;
END_GET
END_PROPERTY

METHOD CyclicLogic
VAR
	i : UINT;
END_VAR
IF NOT Initialized THEN
	Initialize();
	RETURN;
END_IF

IF Simulated THEN
	_Busy		 := FALSE;
	_Error		 := FALSE;
	_ErrorId	 := 0;
	_ErrorSource := E_EcErrorSource.None;
ELSE
	IF NOT _Busy THEN
		IF (LastChangeCount <> EcMaster.ChangeCount) THEN
			RunSlaveDiag := TRUE;
		ELSIF ((EcMaster.CfgSlaveCount <> EcMaster.SlaveCount) AND (LastSlaveCount <> EcMaster.SlaveCount)) THEN
			RunSlaveDiag := TRUE;
		ELSIF FramesWcStatesOk() <> LastFramesWcStatesOk THEN
			RunSlaveDiag := TRUE;
		END_IF

		IF RunSlaveDiag THEN
			LastChangeCount		 := EcMaster.ChangeCount;
			LastSlaveCount		 := EcMaster.SlaveCount;
			LastFramesWcStatesOk := FramesWcStatesOk();
		END_IF
	END_IF

	MasterState();
	SlaveState();
	FOR i := 0 TO (SYNC_UNITS - 1) DO
		SyncUnit[i].CyclicLogic();
	END_FOR

	_Busy := SlaveSequence <> 0;
END_IF

(* Only CoE transfers in flight are serviced; idle io devices cost nothing per cycle. *)
ServiceCoeTransfers();
END_METHOD

// Leaves the slave evaluation: assigns the sync units once they resolved their slave lists, otherwise idles.
METHOD PRIVATE EndDiagnosticPass
IF NOT SyncUnitsAssigned AND_THEN SyncUnitsResolved() THEN
	SyncUnitScan  := 0;
	ScanIndex	  := 0;
	SlaveSequence := 40;
ELSE
	SlaveSequence := 0;
END_IF
END_METHOD

{attribute 'monitoring' := 'call'}
PROPERTY Error : BOOL
GET
Error := _Error;
END_GET
END_PROPERTY

// Raw code of ErrorSource: DevState word (Master), slave index (Slave), ADS error id (Ads), step (Sequence).
{attribute 'monitoring' := 'call'}
PROPERTY ErrorId : UDINT
GET
ErrorId := _ErrorId;
END_GET
END_PROPERTY

{attribute 'monitoring' := 'call'}
PROPERTY ErrorSource : E_EcErrorSource
GET
ErrorSource := _ErrorSource;
END_GET
END_PROPERTY

// Raises the slave events for one configured slave. TRUE when a fault was latched (Error, ErrorSource.Slave).
METHOD PROTECTED EvaluateSlave : BOOL
VAR_INPUT
	Index : UINT;
END_VAR

VAR
	DiagByte : BYTE;
END_VAR
IF SlaveTopologyInfo[Index].nStatusBits.4 THEN
	RETURN; // member of a hot connect group: absence or a non-OP state is not a fault
END_IF

DiagByte := SlavesState[Index].deviceState AND 16#0F;
IF DiagByte <> EC_DEVICE_STATE_OP THEN
	IF SlavesState[Index].deviceState.7 THEN // slave is disabled - warning only
		IF EventProvider <> 0 THEN
			EventProvider.RaiseEtherCatDiagnosticEvent(E_EtherCatMaster.SlaveDisabled, ConfiguredSlaveInfo[Index].sName);
		END_IF
	ELSE
		IF EventProvider <> 0 THEN
			EventProvider.RaiseEtherCatDiagnosticEvent(E_EtherCatMaster.SlaveError, ConfiguredSlaveInfo[Index].sName, LookupSlaveState(Index));
		END_IF

		SetError(E_EcErrorSource.Slave, Index);
		EvaluateSlave := TRUE;
		RETURN;
	END_IF
END_IF

DiagByte := SlavesState[Index].linkState AND 16#0F;
IF DiagByte <> EC_LINK_STATE_OK THEN
	IF EventProvider <> 0 THEN
		EventProvider.RaiseEtherCatDiagnosticEvent(E_EtherCatMaster.SlaveError, ConfiguredSlaveInfo[Index].sName, LookupSlaveState(Index));
	END_IF

	SetError(E_EcErrorSource.Slave, Index);
	EvaluateSlave := TRUE;
END_IF
END_METHOD

// Latches the error, logs Message and parks the init sequence in step 999.
METHOD PRIVATE FailInit
VAR_INPUT
	Source	: E_EcErrorSource;
	ErrorId : UDINT;
	Message : T_MaxString;
END_VAR
SetError(Source, ErrorId);
Trace.LogMessage(Name, Message);
InitSequenceState := 999;
END_METHOD

// Latches the error and aborts the running diagnostic sequence.
METHOD PRIVATE FailSequence
VAR_INPUT
	Source	: E_EcErrorSource;
	ErrorId : UDINT;
END_VAR
SetError(Source, ErrorId);
SlaveSequence := 0;
END_METHOD

(*FB_Init is always available implicitly and it is used primarily for initialization.
The return value is not evaluated. For a specific influence, you can also declare the
methods explicitly and provide additional code there with the standard initialization
code. You can evaluate the return value.*)
METHOD FB_Init : BOOL
VAR_INPUT
	(* TRUE: the retain variables are initialized (reset warm / reset cold)*)
	bInitRetains : BOOL;

	(* TRUE: the instance will be copied to the copy code afterward (online change)   *)
	bInCopyCode		: BOOL;
	Name			: T_MaxString;
	EcStartupCycles : UINT;
END_VAR
THIS^.EcStartupCycles := EcStartupCycles;
END_METHOD

METHOD PROTECTED FramesWcStatesOk : BOOL
VAR
	i : UDINT;
END_VAR
FramesWcStatesOk := TRUE;
IF GetMasterFrameCount.nFrames = 0 THEN
	RETURN;
END_IF

FOR i := 0 TO (MIN(GetMasterFrameCount.nFrames, FRAMES) - 1) DO
	IF FrmXWcState[i] <> 0 THEN
		FramesWcStatesOk := FALSE;
		EXIT;
	END_IF
END_FOR
END_METHOD

// O(1) through the address map. Returns the null device (and logs a warning) for unknown addresses.
METHOD GetIoDeviceByAddr : I_EcIoDevice
VAR_INPUT
	Addr : WORD;
END_VAR

VAR
	Idx : DINT;
END_VAR
IF NOT Initialized THEN
	GetIoDeviceByAddr := NullIoDevice;
	RETURN;
END_IF

Idx := GetSlaveIndexByAddr(WORD_TO_UINT(Addr));
IF Idx >= 0 THEN
	GetIoDeviceByAddr := IoDevice[Idx];
ELSE
	Trace.LogMessage(Name, CONCAT('GetIoDeviceByAddr: no configured slave at address ', TO_STRING(WORD_TO_UINT(Addr))));
	GetIoDeviceByAddr := NullIoDevice;
END_IF
END_METHOD

// Linear search over the configured slaves: call once and keep the result.
// Returns the null device (and logs a warning) if no slave carries that name.
METHOD GetIoDeviceByName : I_EcIoDevice
VAR_INPUT
	Name : STRING(31);
END_VAR

VAR
	i : UINT;
END_VAR
IF NOT Initialized THEN
	GetIoDeviceByName := NullIoDevice;
	RETURN;
END_IF

i := 0;
WHILE i < SlaveCountUsed DO
	IF IoDevice[i].Name = Name THEN
		GetIoDeviceByName := IoDevice[i];
		RETURN;
	END_IF
	i := i + 1;
END_WHILE

Trace.LogMessage(THIS^.Name, CONCAT('GetIoDeviceByName: no configured slave named ', Name));
GetIoDeviceByName := NullIoDevice;
END_METHOD

// Configured slave index (0-based) of the slave with EtherCAT address Addr, -1 if none.
// O(1) for the dense range FIRST_SLAVE_ADDR .. FIRST_SLAVE_ADDR + MAX_EC_SLAVES, linear search otherwise.
METHOD GetSlaveIndexByAddr : DINT
VAR_INPUT
	Addr : UINT;
END_VAR

VAR
	i : UINT;
END_VAR
GetSlaveIndexByAddr := -1;

IF (Addr >= FIRST_SLAVE_ADDR) AND_THEN ((Addr - FIRST_SLAVE_ADDR) <= MAX_EC_SLAVES) THEN
	IF AddrToIndex[Addr - FIRST_SLAVE_ADDR] <> 0 THEN
		GetSlaveIndexByAddr := AddrToIndex[Addr - FIRST_SLAVE_ADDR] - 1;
	END_IF
	RETURN; // the map is complete for this range
END_IF

(* Addresses outside the dense range (assigned by the user): linear search. *)
i := 0;
WHILE i < SlaveCountUsed DO
	IF ConfiguredSlaveInfo[i].nAddr = Addr THEN
		GetSlaveIndexByAddr := i;
		RETURN;
	END_IF
	i := i + 1;
END_WHILE
END_METHOD

// I_EcSlaveRegistry: name of the configured slave at Index, '' if Index is out of range.
METHOD GetSlaveName : STRING
VAR_INPUT
	Index : UINT;
END_VAR
IF Index < SlaveCountUsed THEN
	GetSlaveName := ConfiguredSlaveInfo[Index].sName;
END_IF
END_METHOD

// Init sequence: local AMS Net ID (0) - configured slaves (10) - topology (20) - frame count (30) -
// sync units (40) - startup cycles, io device wiring and address map (50). Step 999 = failed, see trace.
METHOD Initialize
VAR_INST
	GetLocalAmsNetId : FB_GetLocalAmsNetId;
	StartCycles		 : UINT;
END_VAR

VAR
	i : UDINT;
	k : UINT;
END_VAR
IF NOT _Error AND NOT Simulated THEN
	IF F_GetMappingStatus(ADR(EcMaster.AmsNetID), SIZEOF(EcMaster.AmsNetID)) = EplcMappingStatus.MS_Unmapped THEN
		FailInit(E_EcErrorSource.Sequence, InitSequenceState, 'Init Failed - EcMaster.AmsNetID not mapped to the EtherCAT master!');
	ELSIF F_GetMappingStatus(ADR(EcMaster.DevID), SIZEOF(EcMaster.DevID)) = EplcMappingStatus.MS_Unmapped THEN
		FailInit(E_EcErrorSource.Sequence, InitSequenceState, 'Init Failed - EcMaster.DevID not mapped to the EtherCAT master!');
	ELSIF F_GetMappingStatus(ADR(EcMaster.DevState), SIZEOF(EcMaster.DevState)) = EplcMappingStatus.MS_Unmapped THEN
		FailInit(E_EcErrorSource.Sequence, InitSequenceState, 'Init Failed - EcMaster.DevState not mapped to the EtherCAT master!');
	ELSIF F_GetMappingStatus(ADR(EcMaster.ChangeCount), SIZEOF(EcMaster.ChangeCount)) = EplcMappingStatus.MS_Unmapped THEN
		FailInit(E_EcErrorSource.Sequence, InitSequenceState, 'Init Failed - EcMaster.ChangeCount not mapped to the EtherCAT master!');
	ELSIF F_GetMappingStatus(ADR(EcMaster.SlaveCount), SIZEOF(EcMaster.SlaveCount)) = EplcMappingStatus.MS_Unmapped THEN
		FailInit(E_EcErrorSource.Sequence, InitSequenceState, 'Init Failed - EcMaster.SlaveCount not mapped to the EtherCAT master!');
	ELSIF F_GetMappingStatus(ADR(EcMaster.CfgSlaveCount), SIZEOF(EcMaster.CfgSlaveCount)) = EplcMappingStatus.MS_Unmapped THEN
		FailInit(E_EcErrorSource.Sequence, InitSequenceState, 'Init Failed - EcMaster.CfgSlaveCount not mapped to the EtherCAT master!');
	END_IF
END_IF

IF _Error THEN
	RETURN;
END_IF

IF Simulated THEN
	FOR i := 0 TO (SYNC_UNITS - 1) DO
		SyncUnit[i].EventProvider := EventProvider;
		SyncUnit[i].Simulated	  := Simulated;
		SyncUnit[i].Initialize();
		IF NOT SyncUnit[i].Initialized THEN
			RETURN;
		END_IF
	END_FOR

	_Initialized := TRUE;
	RETURN;
END_IF

GetLocalAmsNetId(tTimeOut := T#1S);
_MasterAmsNetId := F_CreateAmsNetId(EcMaster.AmsNetID);
GetMasterFrameCount(sNetId := _MasterAmsNetId, tTimeout := ADS_TIMEOUT);
GetConfiguredSlaves(sNetId				:= _MasterAmsNetId,
					pArrEcConfSlaveInfo := ADR(ConfiguredSlaveInfo),
					cbBufLen			:= SlaveCountUsed * SIZEOF(ConfiguredSlaveInfo[0]),
					tTimeout			:= ADS_TIMEOUT);
GetSlaveTopologyInfo(sNetId	  := _MasterAmsNetId,
					 pAddrBuf := ADR(SlaveTopologyInfo),
					 cbBufLen := TopologyBufLen(),
					 tTimeout := ADS_TIMEOUT);

CASE InitSequenceState OF
	0: (* local AMS Net ID *)
		GetLocalAmsNetId.bExecute := TRUE;
		WaitCycles				  := 0;
		NextMinorStep(InitSequenceState);

	1:
		IF GetLocalAmsNetId.bBusy THEN
			IF AdsWatchdogExpired(ADS_WAIT_CYCLES) THEN
				GetLocalAmsNetId.bExecute := FALSE;
				FailInit(E_EcErrorSource.Ads, ERROR_ADS_TIMEOUT, 'Init Failed - GetLocalAmsNetId timed out!');
			END_IF
		ELSIF GetLocalAmsNetId.bError THEN
			GetLocalAmsNetId.bExecute := FALSE;
			FailInit(E_EcErrorSource.Ads, GetLocalAmsNetId.nErrId, 'Init Failed - GetLocalAmsNetId!');
		ELSE
			GetLocalAmsNetId.bExecute := FALSE;
			_LocalAmsNetId			  := GetLocalAmsNetId.AddrString;
			WaitCycles				  := 0;
			NextStep(InitSequenceState);
		END_IF

	10: (* configured slaves, read sized to the configured count *)
		IF EcMaster.CfgSlaveCount = 0 THEN
			IF AdsWatchdogExpired(ADS_WAIT_CYCLES) THEN
				FailInit(E_EcErrorSource.Sequence, InitSequenceState, 'Init Failed - EcMaster.CfgSlaveCount stays 0: no slaves configured or EcMaster not linked!');
			END_IF
			RETURN;
		END_IF

		IF EcMaster.CfgSlaveCount > (MAX_EC_SLAVES + 1) THEN
			FailInit(E_EcErrorSource.Sequence, EcMaster.CfgSlaveCount, 'Init Failed - more slaves configured than EtherCatParameter.MAX_EC_SLAVES + 1 can hold!');
			RETURN;
		END_IF

		SlaveCountUsed				 := EcMaster.CfgSlaveCount;
		GetConfiguredSlaves.bExecute := TRUE;
		WaitCycles					 := 0;
		NextMinorStep(InitSequenceState);

	11:
		IF GetConfiguredSlaves.bBusy THEN
			IF AdsWatchdogExpired(INIT_WAIT_CYCLES) THEN
				GetConfiguredSlaves.bExecute := FALSE;
				FailInit(E_EcErrorSource.Ads, ERROR_ADS_TIMEOUT, 'Init Failed - reading the configured EtherCAT slaves timed out!');
			END_IF
		ELSIF GetConfiguredSlaves.bError THEN
			GetConfiguredSlaves.bExecute := FALSE;
			FailInit(E_EcErrorSource.Ads, GetConfiguredSlaves.nErrorId, 'Init Failed - configured EtherCAT slaves could not be read - check linking of the EtherCAT master FB!');
		ELSE
			GetConfiguredSlaves.bExecute := FALSE;
			WaitCycles					 := 0;
			NextStep(InitSequenceState);
		END_IF

	20: (* topology: the hot connect flags are needed by the slave evaluation and the sync units *)
		GetSlaveTopologyInfo.bExecute := TRUE;
		WaitCycles					  := 0;
		NextMinorStep(InitSequenceState);

	21:
		IF GetSlaveTopologyInfo.bBusy THEN
			IF AdsWatchdogExpired(INIT_WAIT_CYCLES) THEN
				GetSlaveTopologyInfo.bExecute := FALSE;
				FailInit(E_EcErrorSource.Ads, ERROR_ADS_TIMEOUT, 'Init Failed - reading the EtherCAT topology timed out!');
			END_IF
		ELSIF GetSlaveTopologyInfo.bError THEN
			GetSlaveTopologyInfo.bExecute := FALSE;
			FailInit(E_EcErrorSource.Ads, GetSlaveTopologyInfo.nErrId, 'Init Failed - EtherCAT topology could not be read!');
		ELSE
			GetSlaveTopologyInfo.bExecute := FALSE;
			WaitCycles					  := 0;
			NextStep(InitSequenceState);
		END_IF

	30: (* frame count *)
		GetMasterFrameCount.bExecute := TRUE;
		WaitCycles					 := 0;
		NextMinorStep(InitSequenceState);

	31:
		IF GetMasterFrameCount.bBusy THEN
			IF AdsWatchdogExpired(ADS_WAIT_CYCLES) THEN
				GetMasterFrameCount.bExecute := FALSE;
				FailInit(E_EcErrorSource.Ads, ERROR_ADS_TIMEOUT, 'Init Failed - reading the EtherCAT frame count timed out!');
			END_IF
		ELSIF GetMasterFrameCount.bError THEN
			GetMasterFrameCount.bExecute := FALSE;
			FailInit(E_EcErrorSource.Ads, GetMasterFrameCount.nErrId, 'Init Failed - configured EtherCAT frames could not be read!');
		ELSE
			GetMasterFrameCount.bExecute := FALSE;
			IF GetMasterFrameCount.nFrames = 0 THEN
				FailInit(E_EcErrorSource.Sequence, InitSequenceState, 'Init Failed - the EtherCAT master reports no cyclic frames!');
				RETURN;
			END_IF

			IF GetMasterFrameCount.nFrames > FRAMES THEN
				FailInit(E_EcErrorSource.Sequence, GetMasterFrameCount.nFrames, 'Init Failed - increase the FRAMES generic parameter and link FrmXWcState[x] to the master!');
				RETURN;
			END_IF

			FOR i := 0 TO (GetMasterFrameCount.nFrames - 1) DO
				IF F_GetMappingStatus(ADR(FrmXWcState[i]), SIZEOF(FrmXWcState[i])) = EplcMappingStatus.MS_Unmapped THEN
					FailInit(E_EcErrorSource.Sequence, i, 'Init Failed - FrmXWcState[x] not mapped to the EtherCAT master!');
					RETURN;
				END_IF
			END_FOR

			NextStep(InitSequenceState);
		END_IF

	40: (* sync units *)
		FOR i := 0 TO (SYNC_UNITS - 1) DO
			SyncUnit[i].EventProvider := EventProvider;
			SyncUnit[i].Initialize();
			IF SyncUnit[i].Error THEN
				FailInit(E_EcErrorSource.Sequence, i, 'Init Failed - a sync unit could not be initialised (see its trace message)!');
				RETURN;
			END_IF

			IF NOT SyncUnit[i].Initialized THEN
				RETURN;
			END_IF
		END_FOR

		NextStep(InitSequenceState);

	50: (* let the master settle, then build the address map *)
		StartCycles := StartCycles + 1;
		IF StartCycles >= EcStartupCycles THEN
			BuildAddrToIndex();
			ScanIndex := 0;
			NextMinorStep(InitSequenceState);
		END_IF

	51: (* wire the io devices, SLAVES_PER_CYCLE per cycle *)
		FOR k := 1 TO SLAVES_PER_CYCLE DO
			IF ScanIndex >= SlaveCountUsed THEN
				EXIT;
			END_IF

			IoDevice[ScanIndex].AmsNetId	  := EcMaster.AmsNetID;
			IoDevice[ScanIndex].Name		  := ConfiguredSlaveInfo[ScanIndex].sName;
			IoDevice[ScanIndex].State		  REF= SlavesState[ScanIndex];
			IoDevice[ScanIndex].Configuration REF= ConfiguredSlaveInfo[ScanIndex];
			IoDevice[ScanIndex].CoeScheduler  := THIS^;
			ScanIndex						  := ScanIndex + 1;
		END_FOR

		IF ScanIndex >= SlaveCountUsed THEN
			_Initialized := TRUE;
		END_IF

	999: (* Fail - look at the trace message in the ADS log *)
END_CASE
END_METHOD

{attribute 'monitoring' := 'call'}
PROPERTY Initialized : BOOL
GET
Initialized := _Initialized;
END_GET
SET
_Initialized := Initialized;
END_SET
END_PROPERTY

// I_EcSlaveRegistry: TRUE if the configured slave at Index belongs to a hot connect group
// (topology status bits 4 or 5, read once in Initialize). FALSE if Index is out of range.
METHOD IsHotConnectMember : BOOL
VAR_INPUT
	Index : UINT;
END_VAR
IF Index < SlaveCountUsed THEN
	IsHotConnectMember := SlaveTopologyInfo[Index].nStatusBits.4 OR SlaveTopologyInfo[Index].nStatusBits.5;
END_IF
END_METHOD

{attribute 'monitoring' := 'call'}
PROPERTY LocalAmsNetId : T_AmsNetId
GET
LocalAmsNetId := _LocalAmsNetId;
END_GET
END_PROPERTY

METHOD PROTECTED LookupMasterState : STRING
VAR_INPUT
	State : UINT;
END_VAR
IF State.0 THEN
	LookupMasterState := 'Link error';
ELSIF State.1 THEN
	LookupMasterState := 'I/O locked after link error (I/O reset required)';
ELSIF State.2 THEN
	LookupMasterState := 'Link error (redundancy adapter)';
ELSIF State.3 THEN
	LookupMasterState := 'Missing one frame (redundancy mode)';
ELSIF State.4 THEN
	LookupMasterState := 'Out of send resources (I/O reset required)';
ELSIF State.5 THEN
	LookupMasterState := 'Watchdog triggered';
ELSIF State.6 THEN
	LookupMasterState := 'Ethernet driver (miniport) NOT found';
ELSIF State.7 THEN
	LookupMasterState := 'I/O reset active';
ELSIF State.8 THEN
	LookupMasterState := 'At least one device in INIT state';
ELSIF State.9 THEN
	LookupMasterState := 'At least one device in PRE-OP state';
ELSIF State.10 THEN
	LookupMasterState := 'At least one device in SAFE-OP state';
ELSIF State.11 THEN
	LookupMasterState := 'At least one device indicates an error state';
ELSIF State.12 THEN
	LookupMasterState := 'DC not in sync';
ELSE
	LookupMasterState := 'State not found';
END_IF
END_METHOD

METHOD PROTECTED LookupSlaveState : STRING
VAR_INPUT
	Slave : UINT;
END_VAR

VAR_INST
	DiagByte	: BYTE;
	BitMaskDiag : BYTE := 16#0F;
END_VAR
(* State *)
BitMaskDiag := 16#0F;
DiagByte	:= SlavesState[Slave].deviceState AND BitMaskDiag;
CASE DiagByte OF
	EC_DEVICE_STATE_INIT:
		LookupSlaveState := 'Init';

	EC_DEVICE_STATE_PREOP:
		LookupSlaveState := 'Pre-op';

	EC_DEVICE_STATE_BOOTSTRAP:
		LookupSlaveState := 'Boot';

	EC_DEVICE_STATE_SAFEOP:
		LookupSlaveState := 'Safe-op';

	EC_DEVICE_STATE_OP:
		LookupSlaveState := 'OP';

ELSE
	LookupSlaveState := '';
END_CASE

(* Additional State Bits *)
IF SlavesState[Slave].deviceState.4 THEN // EC_DEVICE_STATE_ERROR
	LookupSlaveState := CONCAT(LookupSlaveState, ' - ');
	LookupSlaveState := CONCAT(LookupSlaveState, 'State machine error in the EtherCAT slave');
END_IF

IF SlavesState[Slave].deviceState.5 THEN // EC_DEVICE_STATE_INVALID_VPRS
	LookupSlaveState := CONCAT(LookupSlaveState, ' - ');
	LookupSlaveState := CONCAT(LookupSlaveState, 'Invalid vendor ID');
END_IF

IF SlavesState[Slave].deviceState.6 THEN // EC_DEVICE_STATE_INITCMD_ERROR
	LookupSlaveState := CONCAT(LookupSlaveState, ' - ');
	LookupSlaveState := CONCAT(LookupSlaveState, 'Error during sending of initialization commands');
END_IF

IF SlavesState[Slave].deviceState.7 THEN // EC_DEVICE_STATE_DISABLED
	LookupSlaveState := CONCAT(LookupSlaveState, ' - ');
	LookupSlaveState := CONCAT(LookupSlaveState, 'Slave is disabled');
END_IF

//_____________________________________________________________________________________________________

(* Link States *)
IF SlavesState[Slave].linkState.0 THEN // EC_LINK_STATE_NOT_PRESENT
	LookupSlaveState := CONCAT(LookupSlaveState, ' - ');
	LookupSlaveState := CONCAT(LookupSlaveState, 'No EtherCAT communication with the EtherCAT slave');
END_IF

IF SlavesState[Slave].linkState.1 THEN // EC_LINK_STATE_LINK_WITHOUT_COMM
	LookupSlaveState := CONCAT(LookupSlaveState, ' - ');
	LookupSlaveState := CONCAT(LookupSlaveState, 'Error AT port X');
END_IF

IF SlavesState[Slave].linkState.2 THEN // EC_LINK_STATE_MISSING_LINK
	LookupSlaveState := CONCAT(LookupSlaveState, ' - ');
	LookupSlaveState := CONCAT(LookupSlaveState, 'Missing link AT port X');
END_IF

IF SlavesState[Slave].linkState.3 THEN // EC_LINK_STATE_ADDITIONAL_LINK
	LookupSlaveState := CONCAT(LookupSlaveState, ' - ');
	LookupSlaveState := CONCAT(LookupSlaveState, 'Additional link AT port X');
END_IF

(* Additional State Bits *)
IF SlavesState[Slave].linkState.4 THEN // EC_LINK_STATE_PORT_A
	LookupSlaveState := CONCAT(LookupSlaveState, ' - ');
	LookupSlaveState := CONCAT(LookupSlaveState, 'Port 0');
END_IF

IF SlavesState[Slave].linkState.5 THEN // EC_LINK_STATE_PORT_B
	LookupSlaveState := CONCAT(LookupSlaveState, ' - ');
	LookupSlaveState := CONCAT(LookupSlaveState, 'Port 1');
END_IF

IF SlavesState[Slave].linkState.6 THEN // EC_LINK_STATE_PORT_C
	LookupSlaveState := CONCAT(LookupSlaveState, ' - ');
	LookupSlaveState := CONCAT(LookupSlaveState, 'Port 2');
END_IF

IF SlavesState[Slave].linkState.7 THEN // EC_LINK_STATE_PORT_D
	LookupSlaveState := CONCAT(LookupSlaveState, ' - ');
	LookupSlaveState := CONCAT(LookupSlaveState, 'Port 3');
END_IF
END_METHOD

// Enters the configured slave Index into the address map if its address lies in the dense range.
METHOD PROTECTED MapSlaveAddress
VAR_INPUT
	Index : UINT;
END_VAR

VAR
	Addr : UINT;
END_VAR
Addr := ConfiguredSlaveInfo[Index].nAddr;
IF (Addr >= FIRST_SLAVE_ADDR) AND_THEN ((Addr - FIRST_SLAVE_ADDR) <= MAX_EC_SLAVES) THEN
	AddrToIndex[Addr - FIRST_SLAVE_ADDR] := Index + 1;
END_IF
END_METHOD

{attribute 'monitoring' := 'call'}
PROPERTY MasterAmsNetId : T_AmsNetId
GET
MasterAmsNetId := _MasterAmsNetId;
END_GET
END_PROPERTY

// Raises one MasterError event per DevState change while slaves are missing. TRUE when an error was latched.
METHOD PROTECTED MasterState : BOOL
VAR_INPUT
END_VAR
IF LastMasterState = EcMaster.DevState THEN
	RETURN;
END_IF

LastMasterState := EcMaster.DevState;

IF (EcMaster.DevState <> 0) AND (EcMaster.SlaveCount < EcMaster.CfgSlaveCount) THEN
	IF EventProvider <> 0 THEN
		EventProvider.RaiseEtherCatDiagnosticEvent(E_EtherCatMaster.MasterError, LookupMasterState(EcMaster.DevState));
	END_IF

	SetError(E_EcErrorSource.Master, EcMaster.DevState);
	MasterState := TRUE;
END_IF
END_METHOD

// I_CoeTransferScheduler: adds a CoE transfer to the set serviced by CyclicLogic (idempotent).
METHOD Register : BOOL
VAR_INPUT
	Transfer : I_CoeTransfer;
END_VAR

VAR
	i : UINT;
END_VAR
IF Transfer = 0 THEN
	RETURN;
END_IF

i := 0;
WHILE i < ActiveCoeCount DO
	IF ActiveCoe[i] = Transfer THEN
		Register := TRUE;
		RETURN;
	END_IF
	i := i + 1;
END_WHILE

IF ActiveCoeCount > MAX_EC_SLAVES THEN
	RETURN; // full
END_IF

ActiveCoe[ActiveCoeCount] := Transfer;
ActiveCoeCount			  := ActiveCoeCount + 1;
Register				  := TRUE;
END_METHOD

METHOD RegisterEventProvider
VAR_INPUT
	EventProvider : I_EtherCatDiagnosticEventProvider;
END_VAR
THIS^.EventProvider := EventProvider;
END_METHOD

METHOD Reset
IF EventProvider <> 0 THEN
	EventProvider.Reset();
END_IF

LastMasterState				  := 0;
LastChangeCount				  := 0;
LastSlaveCount				  := 0;
LastFramesWcStatesOk		  := FALSE;
_Error						  := FALSE;
_ErrorId					  := 0;
_ErrorSource				  := E_EcErrorSource.None;
SlaveSequence				  := 0;
RunSlaveDiag				  := FALSE;
GetAllSlaveStates.bExecute	  := FALSE;
GetSlaveTopologyInfo.bExecute := FALSE;
END_METHOD

